//     PlcTask Outputs/GVL_iXlinker.EtherCAT_Master_EKxxxx.Beckhoff_EKx9xx.Beckhoff_EKx9xxEK1122.A_0006_EK1960_2600_0021.Module_2_FSOUT.Outputs.Relais_Module_Channel_1_Standard_Output_X4_1_X4_5 <-> Module 2 (FSOUT)/Outputs/Relais Module.Channel 1.Standard Output (X4.1, X4.5)
//     PlcTask Outputs/GVL_iXlinker.EtherCAT_Master_EKxxxx.Beckhoff_EKx9xx.Beckhoff_EKx9xxEK1122.A_0006_EK1960_2600_0021.Module_2_FSOUT.Outputs.Relais_Module_Channel_2_Standard_Output_X4_2_X4_6 <-> Module 2 (FSOUT)/Outputs/Relais Module.Channel 2.Standard Output (X4.2, X4.6)
//     PlcTask Outputs/GVL_iXlinker.EtherCAT_Master_EKxxxx.Beckhoff_EKx9xx.Beckhoff_EKx9xxEK1122.A_0006_EK1960_2600_0021.Module_2_FSOUT.Outputs.Relais_Module_Channel_3_Standard_Output_X4_3_X4_7 <-> Module 2 (FSOUT)/Outputs/Relais Module.Channel 3.Standard Output (X4.3, X4.7)
//     PlcTask Outputs/GVL_iXlinker.EtherCAT_Master_EKxxxx.Beckhoff_EKx9xx.Beckhoff_EKx9xxEK1122.A_0006_EK1960_2600_0021.Module_2_FSOUT.Outputs.Relais_Module_Channel_4_Standard_Output_X4_4_X4_8 <-> Module 2 (FSOUT)/Outputs/Relais Module.Channel 4.Standard Output (X4.4, X4.8)
//     PlcTask Inputs/GVL_iXlinker.EtherCAT_Master_EKxxxx.Beckhoff_EKx9xx.Beckhoff_EKx9xxEK1122.A_0006_EK1960_2600_0021.Module_3_FSLOGIC.FSLOGIC_Inputs.Safe_Logic_State <-> Module 3 (FSLOGIC)/FSLOGIC Inputs/Safe Logic State
//     PlcTask Inputs/GVL_iXlinker.EtherCAT_Master_EKxxxx.Beckhoff_EKx9xx.Beckhoff_EKx9xxEK1122.A_0006_EK1960_2600_0021.Module_3_FSLOGIC.FSLOGIC_Inputs.Cycle_Counter <-> Module 3 (FSLOGIC)/FSLOGIC Inputs/Cycle Counter
//     PlcTask Inputs/GVL_iXlinker.EtherCAT_Master_EKxxxx.Beckhoff_EKx9xx.Beckhoff_EKx9xxEK1122.A_0006_EK1960_2600_0021.WcState.WcState0 <-> WcState/WcState0
//     PlcTask Inputs/GVL_iXlinker.EtherCAT_Master_EKxxxx.Beckhoff_EKx9xx.Beckhoff_EKx9xxEK1122.A_0006_EK1960_2600_0021.WcState.WcState1 <-> WcState/WcState1
//     PlcTask Inputs/GVL_iXlinker.EtherCAT_Master_EKxxxx.Beckhoff_EKx9xx.Beckhoff_EKx9xxEK1122.A_0006_EK1960_2600_0021.WcState.InputToggle0 <-> WcState/InputToggle0
//     PlcTask Inputs/GVL_iXlinker.EtherCAT_Master_EKxxxx.Beckhoff_EKx9xx.Beckhoff_EKx9xxEK1122.A_0006_EK1960_2600_0021.WcState.InputToggle1 <-> WcState/InputToggle1
//     PlcTask Inputs/GVL_iXlinker.EtherCAT_Master_EKxxxx.Beckhoff_EKx9xx.Beckhoff_EKx9xxEK1122.A_0006_EK1960_2600_0021.InfoData.AdsAddr <-> InfoData/AdsAddr
//     PlcTask Inputs/GVL_iXlinker.EtherCAT_Master_EKxxxx.Beckhoff_EKx9xx.Beckhoff_EKx9xxEK1122.A_0006_EK1960_2600_0021.InfoData.State <-> InfoData/State
//   PLC/PLC Instance <-> EtherCAT Master EKxxxx/Beckhoff EKx9xx/Beckhoff EKx9xxEK1122/A_0007(EK1960-2608-0019)
//     PlcTask Inputs/GVL_iXlinker.EtherCAT_Master_EKxxxx.Beckhoff_EKx9xx.Beckhoff_EKx9xxEK1122.A_0007_EK1960_2608_0019.Module_1_FSoE.FSoE_Inputs.FSOE/FSoE_Command <-> Module 1 (FSoE)/FSoE Inputs/FSOE/FSoE Command
//     PlcTask Inputs/GVL_iXlinker.EtherCAT_Master_EKxxxx.Beckhoff_EKx9xx.Beckhoff_EKx9xxEK1122.A_0007_EK1960_2608_0019.Module_1_FSoE.FSoE_Inputs.FSOE/FSOUT_Module_1_Module_Fault <-> Module 1 (FSoE)/FSoE Inputs/FSOE/FSOUT Module 1.Module Fault
//     PlcTask Inputs/GVL_iXlinker.EtherCAT_Master_EKxxxx.Beckhoff_EKx9xx.Beckhoff_EKx9xxEK1122.A_0007_EK1960_2608_0019.Module_1_FSoE.FSoE_Inputs.FSOE/FSOUT_Module_2_Module_Fault <-> Module 1 (FSoE)/FSoE Inputs/FSOE/FSOUT Module 2.Module Fault
//     PlcTask Inputs/GVL_iXlinker.EtherCAT_Master_EKxxxx.Beckhoff_EKx9xx.Beckhoff_EKx9xxEK1122.A_0007_EK1960_2608_0019.Module_1_FSoE.FSoE_Inputs.FSOE/FSOUT_Module_3_Module_Fault <-> Module 1 (FSoE)/FSoE Inputs/FSOE/FSOUT Module 3.Module Fault
//     PlcTask Inputs/GVL_iXlinker.EtherCAT_Master_EKxxxx.Beckhoff_EKx9xx.Beckhoff_EKx9xxEK1122.A_0007_EK1960_2608_0019.Module_1_FSoE.FSoE_Inputs.FSOE/FSOUT_Module_4_Module_Fault <-> Module 1 (FSoE)/FSoE Inputs/FSOE/FSOUT Module 4.Module Fault
//     PlcTask Inputs/GVL_iXlinker.EtherCAT_Master_EKxxxx.Beckhoff_EKx9xx.Beckhoff_EKx9xxEK1122.A_0007_EK1960_2608_0019.Module_1_FSoE.FSoE_Inputs.FSOE/FSOUT_Module_5_Module_Fault <-> Module 1 (FSoE)/FSoE Inputs/FSOE/FSOUT Module 5.Module Fault
//     PlcTask Inputs/GVL_iXlinker.EtherCAT_Master_EKxxxx.Beckhoff_EKx9xx.Beckhoff_EKx9xxEK1122.A_0007_EK1960_2608_0019.Module_1_FSoE.FSoE_Inputs.FSOE/FSOUT_Module_6_Module_Fault <-> Module 1 (FSoE)/FSoE Inputs/FSOE/FSOUT Module 6.Module Fault
//     PlcTask Inputs/GVL_iXlinker.EtherCAT_Master_EKxxxx.Beckhoff_EKx9xx.Beckhoff_EKx9xxEK1122.A_0007_EK1960_2608_0019.Module_1_FSoE.FSoE_Inputs.FSOE/FSOUT_Relais_Module_Module_Fault <-> Module 1 (FSoE)/FSoE Inputs/FSOE/FSOUT Relais Module.Module Fault
//     PlcTask Inputs/GVL_iXlinker.EtherCAT_Master_EKxxxx.Beckhoff_EKx9xx.Beckhoff_EKx9xxEK1122.A_0007_EK1960_2608_0019.Module_1_FSoE.FSoE_Inputs.FSOE/FSIN_Module_1_Channel_1_Input <-> Module 1 (FSoE)/FSoE Inputs/FSOE/FSIN Module 1.Channel 1.Input
//     PlcTask Inputs/GVL_iXlinker.EtherCAT_Master_EKxxxx.Beckhoff_EKx9xx.Beckhoff_EKx9xxEK1122.A_0007_EK1960_2608_0019.Module_1_FSoE.FSoE_Inputs.FSOE/FSIN_Module_1_Channel_2_Input <-> Module 1 (FSoE)/FSoE Inputs/FSOE/FSIN Module 1.Channel 2.Input
//     PlcTask Inputs/GVL_iXlinker.EtherCAT_Master_EKxxxx.Beckhoff_EKx9xx.Beckhoff_EKx9xxEK1122.A_0007_EK1960_2608_0019.Module_1_FSoE.FSoE_Inputs.FSOE/FSIN_Module_2_Channel_1_Input <-> Module 1 (FSoE)/FSoE Inputs/FSOE/FSIN Module 2.Channel 1.Input
//     PlcTask Inputs/GVL_iXlinker.EtherCAT_Master_EKxxxx.Beckhoff_EKx9xx.Beckhoff_EKx9xxEK1122.A_0007_EK1960_2608_0019.Module_1_FSoE.FSoE_Inputs.FSOE/FSIN_Module_2_Channel_2_Input <-> Module 1 (FSoE)/FSoE Inputs/FSOE/FSIN Module 2.Channel 2.Input
//     PlcTask Inputs/GVL_iXlinker.EtherCAT_Master_EKxxxx.Beckhoff_EKx9xx.Beckhoff_EKx9xxEK1122.A_0007_EK1960_2608_0019.Module_1_FSoE.FSoE_Inputs.FSOE/FSIN_Module_3_Channel_1_Input <-> Module 1 (FSoE)/FSoE Inputs/FSOE/FSIN Module 3.Channel 1.Input
//     PlcTask Inputs/GVL_iXlinker.EtherCAT_Master_EKxxxx.Beckhoff_EKx9xx.Beckhoff_EKx9xxEK1122.A_0007_EK1960_2608_0019.Module_1_FSoE.FSoE_Inputs.FSOE/FSIN_Module_3_Channel_2_Input <-> Module 1 (FSoE)/FSoE Inputs/FSOE/FSIN Module 3.Channel 2.Input
//     PlcTask Inputs/GVL_iXlinker.EtherCAT_Master_EKxxxx.Beckhoff_EKx9xx.Beckhoff_EKx9xxEK1122.A_0007_EK1960_2608_0019.Module_1_FSoE.FSoE_Inputs.FSOE/FSIN_Module_4_Channel_1_Input <-> Module 1 (FSoE)/FSoE Inputs/FSOE/FSIN Module 4.Channel 1.Input
//     PlcTask Inputs/GVL_iXlinker.EtherCAT_Master_EKxxxx.Beckhoff_EKx9xx.Beckhoff_EKx9xxEK1122.A_0007_EK1960_2608_0019.Module_1_FSoE.FSoE_Inputs.FSOE/FSIN_Module_4_Channel_2_Input <-> Module 1 (FSoE)/FSoE Inputs/FSOE/FSIN Module 4.Channel 2.Input
//     PlcTask Inputs/GVL_iXlinker.EtherCAT_Master_EKxxxx.Beckhoff_EKx9xx.Beckhoff_EKx9xxEK1122.A_0007_EK1960_2608_0019.Module_1_FSoE.FSoE_Inputs.FSOE/FSIN_Module_5_Channel_1_Input <-> Module 1 (FSoE)/FSoE Inputs/FSOE/FSIN Module 5.Channel 1.Input
//     PlcTask Inputs/GVL_iXlinker.EtherCAT_Master_EKxxxx.Beckhoff_EKx9xx.Beckhoff_EKx9xxEK1122.A_0007_EK1960_2608_0019.Module_1_FSoE.FSoE_Inputs.FSOE/FSIN_Module_5_Channel_2_Input <-> Module 1 (FSoE)/FSoE Inputs/FSOE/FSIN Module 5.Channel 2.Input
//     PlcTask Inputs/GVL_iXlinker.EtherCAT_Master_EKxxxx.Beckhoff_EKx9xx.Beckhoff_EKx9xxEK1122.A_0007_EK1960_2608_0019.Module_1_FSoE.FSoE_Inputs.FSOE/FSIN_Module_6_Channel_1_Input <-> Module 1 (FSoE)/FSoE Inputs/FSOE/FSIN Module 6.Channel 1.Input
//     PlcTask Inputs/GVL_iXlinker.EtherCAT_Master_EKxxxx.Beckhoff_EKx9xx.Beckhoff_EKx9xxEK1122.A_0007_EK1960_2608_0019.Module_1_FSoE.FSoE_Inputs.FSOE/FSIN_Module_6_Channel_2_Input <-> Module 1 (FSoE)/FSoE Inputs/FSOE/FSIN Module 6.Channel 2.Input
//     PlcTask Inputs/GVL_iXlinker.EtherCAT_Master_EKxxxx.Beckhoff_EKx9xx.Beckhoff_EKx9xxEK1122.A_0007_EK1960_2608_0019.Module_1_FSoE.FSoE_Inputs.FSOE/FSIN_Module_7_Channel_1_Input <-> Module 1 (FSoE)/FSoE Inputs/FSOE/FSIN Module 7.Channel 1.Input
//     PlcTask Inputs/GVL_iXlinker.EtherCAT_Master_EKxxxx.Beckhoff_EKx9xx.Beckhoff_EKx9xxEK1122.A_0007_EK1960_2608_0019.Module_1_FSoE.FSoE_Inputs.FSOE/FSIN_Module_7_Channel_2_Input <-> Module 1 (FSoE)/FSoE Inputs/FSOE/FSIN Module 7.Channel 2.Input
//     PlcTask Inputs/GVL_iXlinker.EtherCAT_Master_EKxxxx.Beckhoff_EKx9xx.Beckhoff_EKx9xxEK1122.A_0007_EK1960_2608_0019.Module_1_FSoE.FSoE_Inputs.FSOE/FSIN_Module_8_Channel_1_Input <-> Module 1 (FSoE)/FSoE Inputs/FSOE/FSIN Module 8.Channel 1.Input
//     PlcTask Inputs/GVL_iXlinker.EtherCAT_Master_EKxxxx.Beckhoff_EKx9xx.Beckhoff_EKx9xxEK1122.A_0007_EK1960_2608_0019.Module_1_FSoE.FSoE_Inputs.FSOE/FSIN_Module_8_Channel_2_Input <-> Module 1 (FSoE)/FSoE Inputs/FSOE/FSIN Module 8.Channel 2.Input
//     PlcTask Inputs/GVL_iXlinker.EtherCAT_Master_EKxxxx.Beckhoff_EKx9xx.Beckhoff_EKx9xxEK1122.A_0007_EK1960_2608_0019.Module_1_FSoE.FSoE_Inputs.FSOE/FSIN_Module_9_Channel_1_Input <-> Module 1 (FSoE)/FSoE Inputs/FSOE/FSIN Module 9.Channel 1.Input
//     PlcTask Inputs/GVL_iXlinker.EtherCAT_Master_EKxxxx.Beckhoff_EKx9xx.Beckhoff_EKx9xxEK1122.A_0007_EK1960_2608_0019.Module_1_FSoE.FSoE_Inputs.FSOE/FSIN_Module_9_Channel_2_Input <-> Module 1 (FSoE)/FSoE Inputs/FSOE/FSIN Module 9.Channel 2.Input
//     PlcTask Inputs/GVL_iXlinker.EtherCAT_Master_EKxxxx.Beckhoff_EKx9xx.Beckhoff_EKx9xxEK1122.A_0007_EK1960_2608_0019.Module_1_FSoE.FSoE_Inputs.FSOE/FSIN_Module_10_Channel_1_Input <-> Module 1 (FSoE)/FSoE Inputs/FSOE/FSIN Module 10.Channel 1.Input
//     PlcTask Inputs/GVL_iXlinker.EtherCAT_Master_EKxxxx.Beckhoff_EKx9xx.Beckhoff_EKx9xxEK1122.A_0007_EK1960_2608_0019.Module_1_FSoE.FSoE_Inputs.FSOE/FSIN_Module_10_Channel_2_Input <-> Module 1 (FSoE)/FSoE Inputs/FSOE/FSIN Module 10.Channel 2.Input
//     PlcTask Inputs/GVL_iXlinker.EtherCAT_Master_EKxxxx.Beckhoff_EKx9xx.Beckhoff_EKx9xxEK1122.A_0007_EK1960_2608_0019.Module_1_FSoE.FSoE_Inputs.FSOE/FSIN_Module_1_Module_Fault <-> Module 1 (FSoE)/FSoE Inputs/FSOE/FSIN Module 1.Module Fault
//     PlcTask Inputs/GVL_iXlinker.EtherCAT_Master_EKxxxx.Beckhoff_EKx9xx.Beckhoff_EKx9xxEK1122.A_0007_EK1960_2608_0019.Module_1_FSoE.FSoE_Inputs.FSOE/FSIN_Module_2_Module_Fault <-> Module 1 (FSoE)/FSoE Inputs/FSOE/FSIN Module 2.Module Fault
//     PlcTask Inputs/GVL_iXlinker.EtherCAT_Master_EKxxxx.Beckhoff_EKx9xx.Beckhoff_EKx9xxEK1122.A_0007_EK1960_2608_0019.Module_1_FSoE.FSoE_Inputs.FSOE/FSIN_Module_3_Module_Fault <-> Module 1 (FSoE)/FSoE Inputs/FSOE/FSIN Module 3.Module Fault
//     PlcTask Inputs/GVL_iXlinker.EtherCAT_Master_EKxxxx.Beckhoff_EKx9xx.Beckhoff_EKx9xxEK1122.A_0007_EK1960_2608_0019.Module_1_FSoE.FSoE_Inputs.FSOE/FSIN_Module_4_Module_Fault <-> Module 1 (FSoE)/FSoE Inputs/FSOE/FSIN Module 4.Module Fault
//     PlcTask Inputs/GVL_iXlinker.EtherCAT_Master_EKxxxx.Beckhoff_EKx9xx.Beckhoff_EKx9xxEK1122.A_0007_EK1960_2608_0019.Module_1_FSoE.FSoE_Inputs.FSOE/FSIN_Module_5_Module_Fault <-> Module 1 (FSoE)/FSoE Inputs/FSOE/FSIN Module 5.Module Fault
//     PlcTask Inputs/GVL_iXlinker.EtherCAT_Master_EKxxxx.Beckhoff_EKx9xx.Beckhoff_EKx9xxEK1122.A_0007_EK1960_2608_0019.Module_1_FSoE.FSoE_Inputs.FSOE/FSIN_Module_6_Module_Fault <-> Module 1 (FSoE)/FSoE Inputs/FSOE/FSIN Module 6.Module Fault
//     PlcTask Inputs/GVL_iXlinker.EtherCAT_Master_EKxxxx.Beckhoff_EKx9xx.Beckhoff_EKx9xxEK1122.A_0007_EK1960_2608_0019.Module_1_FSoE.FSoE_Inputs.FSOE/FSIN_Module_7_Module_Fault <-> Module 1 (FSoE)/FSoE Inputs/FSOE/FSIN Module 7.Module Fault
//     PlcTask Inputs/GVL_iXlinker.EtherCAT_Master_EKxxxx.Beckhoff_EKx9xx.Beckhoff_EKx9xxEK1122.A_0007_EK1960_2608_0019.Module_1_FSoE.FSoE_Inputs.FSOE/FSIN_Module_8_Module_Fault <-> Module 1 (FSoE)/FSoE Inputs/FSOE/FSIN Module 8.Module Fault
//     PlcTask Inputs/GVL_iXlinker.EtherCAT_Master_EKxxxx.Beckhoff_EKx9xx.Beckhoff_EKx9xxEK1122.A_0007_EK1960_2608_0019.Module_1_FSoE.FSoE_Inputs.FSOE/FSoE_CRC_000 <-> Module 1 (FSoE)/FSoE Inputs/FSOE/FSoE CRC 000
//     PlcTask Inputs/GVL_iXlinker.EtherCAT_Master_EKxxxx.Beckhoff_EKx9xx.Beckhoff_EKx9xxEK1122.A_0007_EK1960_2608_0019.Module_1_FSoE.FSoE_Inputs.FSOE/FSoE_CRC_001 <-> Module 1 (FSoE)/FSoE Inputs/FSOE/FSoE CRC 001
//     PlcTask Inputs/GVL_iXlinker.EtherCAT_Master_EKxxxx.Beckhoff_EKx9xx.Beckhoff_EKx9xxEK1122.A_0007_EK1960_2608_0019.Module_1_FSoE.FSoE_Inputs.FSOE/FSoE_CRC_002 <-> Module 1 (FSoE)/FSoE Inputs/FSOE/FSoE CRC 002
//     PlcTask Inputs/GVL_iXlinker.EtherCAT_Master_EKxxxx.Beckhoff_EKx9xx.Beckhoff_EKx9xxEK1122.A_0007_EK1960_2608_0019.Module_1_FSoE.FSoE_Inputs.FSOE/FSIN_Module_9_Module_Fault_1 <-> Module 1 (FSoE)/FSoE Inputs/FSOE/FSIN Module 9.Module Fault 1
//     PlcTask Inputs/GVL_iXlinker.EtherCAT_Master_EKxxxx.Beckhoff_EKx9xx.Beckhoff_EKx9xxEK1122.A_0007_EK1960_2608_0019.Module_1_FSoE.FSoE_Inputs.FSOE/FSIN_Module_9_Module_Fault_2 <-> Module 1 (FSoE)/FSoE Inputs/FSOE/FSIN Module 9.Module Fault 2
//     PlcTask Inputs/GVL_iXlinker.EtherCAT_Master_EKxxxx.Beckhoff_EKx9xx.Beckhoff_EKx9xxEK1122.A_0007_EK1960_2608_0019.Module_1_FSoE.FSoE_Inputs.FSOE/FSIN_Module_10_Module_Fault_1 <-> Module 1 (FSoE)/FSoE Inputs/FSOE/FSIN Module 10.Module Fault 1
//     PlcTask Inputs/GVL_iXlinker.EtherCAT_Master_EKxxxx.Beckhoff_EKx9xx.Beckhoff_EKx9xxEK1122.A_0007_EK1960_2608_0019.Module_1_FSoE.FSoE_Inputs.FSOE/FSIN_Module_10_Module_Fault_2 <-> Module 1 (FSoE)/FSoE Inputs/FSOE/FSIN Module 10.Module Fault 2
//     PlcTask Inputs/GVL_iXlinker.EtherCAT_Master_EKxxxx.Beckhoff_EKx9xx.Beckhoff_EKx9xxEK1122.A_0007_EK1960_2608_0019.Module_1_FSoE.FSoE_Inputs.FSOE/FSoE_Connection_ID <-> Module 1 (FSoE)/FSoE Inputs/FSOE/FSoE Connection ID
//     PlcTask Outputs/GVL_iXlinker.EtherCAT_Master_EKxxxx.Beckhoff_EKx9xx.Beckhoff_EKx9xxEK1122.A_0007_EK1960_2608_0019.Module_1_FSoE.FSoE_Outputs.FSOE/FSoE_Command <-> Module 1 (FSoE)/FSoE Outputs/FSOE/FSoE Command
//     PlcTask Outputs/GVL_iXlinker.EtherCAT_Master_EKxxxx.Beckhoff_EKx9xx.Beckhoff_EKx9xxEK1122.A_0007_EK1960_2608_0019.Module_1_FSoE.FSoE_Outputs.FSOE/FSOUT_Module_1_Channel_1_Output <-> Module 1 (FSoE)/FSoE Outputs/FSOE/FSOUT Module 1.Channel 1.Output
//     PlcTask Outputs/GVL_iXlinker.EtherCAT_Master_EKxxxx.Beckhoff_EKx9xx.Beckhoff_EKx9xxEK1122.A_0007_EK1960_2608_0019.Module_1_FSoE.FSoE_Outputs.FSOE/FSOUT_Module_1_Channel_2_Output <-> Module 1 (FSoE)/FSoE Outputs/FSOE/FSOUT Module 1.Channel 2.Output
//     PlcTask Outputs/GVL_iXlinker.EtherCAT_Master_EKxxxx.Beckhoff_EKx9xx.Beckhoff_EKx9xxEK1122.A_0007_EK1960_2608_0019.Module_1_FSoE.FSoE_Outputs.FSOE/FSOUT_Module_1_Channel_3_Output <-> Module 1 (FSoE)/FSoE Outputs/FSOE/FSOUT Module 1.Channel 3.Output
//     PlcTask Outputs/GVL_iXlinker.EtherCAT_Master_EKxxxx.Beckhoff_EKx9xx.Beckhoff_EKx9xxEK1122.A_0007_EK1960_2608_0019.Module_1_FSoE.FSoE_Outputs.FSOE/FSOUT_Module_1_Channel_4_Output <-> Module 1 (FSoE)/FSoE Outputs/FSOE/FSOUT Module 1.Channel 4.Output
//     PlcTask Outputs/GVL_iXlinker.EtherCAT_Master_EKxxxx.Beckhoff_EKx9xx.Beckhoff_EKx9xxEK1122.A_0007_EK1960_2608_0019.Module_1_FSoE.FSoE_Outputs.FSOE/FSOUT_Module_2_Channel_1_Output <-> Module 1 (FSoE)/FSoE Outputs/FSOE/FSOUT Module 2.Channel 1.Output
//     PlcTask Outputs/GVL_iXlinker.EtherCAT_Master_EKxxxx.Beckhoff_EKx9xx.Beckhoff_EKx9xxEK1122.A_0007_EK1960_2608_0019.Module_1_FSoE.FSoE_Outputs.FSOE/FSOUT_Module_2_Channel_2_Output <-> Module 1 (FSoE)/FSoE Outputs/FSOE/FSOUT Module 2.Channel 2.Output
//     PlcTask Outputs/GVL_iXlinker.EtherCAT_Master_EKxxxx.Beckhoff_EKx9xx.Beckhoff_EKx9xxEK1122.A_0007_EK1960_2608_0019.Module_1_FSoE.FSoE_Outputs.FSOE/FSOUT_Module_2_Channel_3_Output <-> Module 1 (FSoE)/FSoE Outputs/FSOE/FSOUT Module 2.Channel 3.Output
//     PlcTask Outputs/GVL_iXlinker.EtherCAT_Master_EKxxxx.Beckhoff_EKx9xx.Beckhoff_EKx9xxEK1122.A_0007_EK1960_2608_0019.Module_1_FSoE.FSoE_Outputs.FSOE/FSOUT_Module_2_Channel_4_Output <-> Module 1 (FSoE)/FSoE Outputs/FSOE/FSOUT Module 2.Channel 4.Output
//     PlcTask Outputs/GVL_iXlinker.EtherCAT_Master_EKxxxx.Beckhoff_EKx9xx.Beckhoff_EKx9xxEK1122.A_0007_EK1960_2608_0019.Module_1_FSoE.FSoE_Outputs.FSOE/FSOUT_Module_3_Channel_1_Output <-> Module 1 (FSoE)/FSoE Outputs/FSOE/FSOUT Module 3.Channel 1.Output
//     PlcTask Outputs/GVL_iXlinker.EtherCAT_Master_EKxxxx.Beckhoff_EKx9xx.Beckhoff_EKx9xxEK1122.A_0007_EK1960_2608_0019.Module_1_FSoE.FSoE_Outputs.FSOE/FSOUT_Module_3_Channel_2_Output <-> Module 1 (FSoE)/FSoE Outputs/FSOE/FSOUT Module 3.Channel 2.Output
//     PlcTask Outputs/GVL_iXlinker.EtherCAT_Master_EKxxxx.Beckhoff_EKx9xx.Beckhoff_EKx9xxEK1122.A_0007_EK1960_2608_0019.Module_1_FSoE.FSoE_Outputs.FSOE/FSOUT_Module_3_Channel_3_Output <-> Module 1 (FSoE)/FSoE Outputs/FSOE/FSOUT Module 3.Channel 3.Output
//     PlcTask Outputs/GVL_iXlinker.EtherCAT_Master_EKxxxx.Beckhoff_EKx9xx.Beckhoff_EKx9xxEK1122.A_0007_EK1960_2608_0019.Module_1_FSoE.FSoE_Outputs.FSOE/FSOUT_Module_3_Channel_4_Output <-> Module 1 (FSoE)/FSoE Outputs/FSOE/FSOUT Module 3.Channel 4.Output
//     PlcTask Outputs/GVL_iXlinker.EtherCAT_Master_EKxxxx.Beckhoff_EKx9xx.Beckhoff_EKx9xxEK1122.A_0007_EK1960_2608_0019.Module_1_FSoE.FSoE_Outputs.FSOE/FSOUT_Module_4_Channel_1_Output <-> Module 1 (FSoE)/FSoE Outputs/FSOE/FSOUT Module 4.Channel 1.Output
//     PlcTask Outputs/GVL_iXlinker.EtherCAT_Master_EKxxxx.Beckhoff_EKx9xx.Beckhoff_EKx9xxEK1122.A_0007_EK1960_2608_0019.Module_1_FSoE.FSoE_Outputs.FSOE/FSOUT_Module_4_Channel_2_Output <-> Module 1 (FSoE)/FSoE Outputs/FSOE/FSOUT Module 4.Channel 2.Output
//     PlcTask Outputs/GVL_iXlinker.EtherCAT_Master_EKxxxx.Beckhoff_EKx9xx.Beckhoff_EKx9xxEK1122.A_0007_EK1960_2608_0019.Module_1_FSoE.FSoE_Outputs.FSOE/FSOUT_Module_4_Channel_3_Output <-> Module 1 (FSoE)/FSoE Outputs/FSOE/FSOUT Module 4.Channel 3.Output
//     PlcTask Outputs/GVL_iXlinker.EtherCAT_Master_EKxxxx.Beckhoff_EKx9xx.Beckhoff_EKx9xxEK1122.A_0007_EK1960_2608_0019.Module_1_FSoE.FSoE_Outputs.FSOE/FSOUT_Module_4_Channel_4_Output <-> Module 1 (FSoE)/FSoE Outputs/FSOE/FSOUT Module 4.Channel 4.Output
//     PlcTask Outputs/GVL_iXlinker.EtherCAT_Master_EKxxxx.Beckhoff_EKx9xx.Beckhoff_EKx9xxEK1122.A_0007_EK1960_2608_0019.Module_1_FSoE.FSoE_Outputs.FSOE/FSOUT_Module_5_Channel_1_Output <-> Module 1 (FSoE)/FSoE Outputs/FSOE/FSOUT Module 5.Channel 1.Output
//     PlcTask Outputs/GVL_iXlinker.EtherCAT_Master_EKxxxx.Beckhoff_EKx9xx.Beckhoff_EKx9xxEK1122.A_0007_EK1960_2608_0019.Module_1_FSoE.FSoE_Outputs.FSOE/FSOUT_Module_5_Channel_2_Output <-> Module 1 (FSoE)/FSoE Outputs/FSOE/FSOUT Module 5.Channel 2.Output
//     PlcTask Outputs/GVL_iXlinker.EtherCAT_Master_EKxxxx.Beckhoff_EKx9xx.Beckhoff_EKx9xxEK1122.A_0007_EK1960_2608_0019.Module_1_FSoE.FSoE_Outputs.FSOE/FSOUT_Module_5_Channel_3_Output <-> Module 1 (FSoE)/FSoE Outputs/FSOE/FSOUT Module 5.Channel 3.Output
//     PlcTask Outputs/GVL_iXlinker.EtherCAT_Master_EKxxxx.Beckhoff_EKx9xx.Beckhoff_EKx9xxEK1122.A_0007_EK1960_2608_0019.Module_1_FSoE.FSoE_Outputs.FSOE/FSOUT_Module_5_Channel_4_Output <-> Module 1 (FSoE)/FSoE Outputs/FSOE/FSOUT Module 5.Channel 4.Output
//     PlcTask Outputs/GVL_iXlinker.EtherCAT_Master_EKxxxx.Beckhoff_EKx9xx.Beckhoff_EKx9xxEK1122.A_0007_EK1960_2608_0019.Module_1_FSoE.FSoE_Outputs.FSOE/FSOUT_Module_6_Channel_1_Output <-> Module 1 (FSoE)/FSoE Outputs/FSOE/FSOUT Module 6.Channel 1.Output
//     PlcTask Outputs/GVL_iXlinker.EtherCAT_Master_EKxxxx.Beckhoff_EKx9xx.Beckhoff_EKx9xxEK1122.A_0007_EK1960_2608_0019.Module_1_FSoE.FSoE_Outputs.FSOE/FSOUT_Module_6_Channel_2_Output <-> Module 1 (FSoE)/FSoE Outputs/FSOE/FSOUT Module 6.Channel 2.Output
//     PlcTask Outputs/GVL_iXlinker.EtherCAT_Master_EKxxxx.Beckhoff_EKx9xx.Beckhoff_EKx9xxEK1122.A_0007_EK1960_2608_0019.Module_1_FSoE.FSoE_Outputs.FSOE/FSOUT_Module_6_Channel_3_Output <-> Module 1 (FSoE)/FSoE Outputs/FSOE/FSOUT Module 6.Channel 3.Output
//     PlcTask Outputs/GVL_iXlinker.EtherCAT_Master_EKxxxx.Beckhoff_EKx9xx.Beckhoff_EKx9xxEK1122.A_0007_EK1960_2608_0019.Module_1_FSoE.FSoE_Outputs.FSOE/FSOUT_Module_6_Channel_4_Output <-> Module 1 (FSoE)/FSoE Outputs/FSOE/FSOUT Module 6.Channel 4.Output
//     PlcTask Outputs/GVL_iXlinker.EtherCAT_Master_EKxxxx.Beckhoff_EKx9xx.Beckhoff_EKx9xxEK1122.A_0007_EK1960_2608_0019.Module_1_FSoE.FSoE_Outputs.FSOE/FSOUT_Module_1_ErrAck <-> Module 1 (FSoE)/FSoE Outputs/FSOE/FSOUT Module 1.ErrAck
//     PlcTask Outputs/GVL_iXlinker.EtherCAT_Master_EKxxxx.Beckhoff_EKx9xx.Beckhoff_EKx9xxEK1122.A_0007_EK1960_2608_0019.Module_1_FSoE.FSoE_Outputs.FSOE/FSOUT_Module_2_ErrAck <-> Module 1 (FSoE)/FSoE Outputs/FSOE/FSOUT Module 2.ErrAck
//     PlcTask Outputs/GVL_iXlinker.EtherCAT_Master_EKxxxx.Beckhoff_EKx9xx.Beckhoff_EKx9xxEK1122.A_0007_EK1960_2608_0019.Module_1_FSoE.FSoE_Outputs.FSOE/FSOUT_Module_3_ErrAck <-> Module 1 (FSoE)/FSoE Outputs/FSOE/FSOUT Module 3.ErrAck
//     PlcTask Outputs/GVL_iXlinker.EtherCAT_Master_EKxxxx.Beckhoff_EKx9xx.Beckhoff_EKx9xxEK1122.A_0007_EK1960_2608_0019.Module_1_FSoE.FSoE_Outputs.FSOE/FSOUT_Module_4_ErrAck <-> Module 1 (FSoE)/FSoE Outputs/FSOE/FSOUT Module 4.ErrAck
//     PlcTask Outputs/GVL_iXlinker.EtherCAT_Master_EKxxxx.Beckhoff_EKx9xx.Beckhoff_EKx9xxEK1122.A_0007_EK1960_2608_0019.Module_1_FSoE.FSoE_Outputs.FSOE/FSOUT_Module_5_ErrAck <-> Module 1 (FSoE)/FSoE Outputs/FSOE/FSOUT Module 5.ErrAck
//     PlcTask Outputs/GVL_iXlinker.EtherCAT_Master_EKxxxx.Beckhoff_EKx9xx.Beckhoff_EKx9xxEK1122.A_0007_EK1960_2608_0019.Module_1_FSoE.FSoE_Outputs.FSOE/FSOUT_Module_6_ErrAck <-> Module 1 (FSoE)/FSoE Outputs/FSOE/FSOUT Module 6.ErrAck
//     PlcTask Outputs/GVL_iXlinker.EtherCAT_Master_EKxxxx.Beckhoff_EKx9xx.Beckhoff_EKx9xxEK1122.A_0007_EK1960_2608_0019.Module_1_FSoE.FSoE_Outputs.FSOE/FSoE_CRC_000 <-> Module 1 (FSoE)/FSoE Outputs/FSOE/FSoE CRC 000
//     PlcTask Outputs/GVL_iXlinker.EtherCAT_Master_EKxxxx.Beckhoff_EKx9xx.Beckhoff_EKx9xxEK1122.A_0007_EK1960_2608_0019.Module_1_FSoE.FSoE_Outputs.FSOE/FSoE_CRC_001 <-> Module 1 (FSoE)/FSoE Outputs/FSOE/FSoE CRC 001
//     PlcTask Outputs/GVL_iXlinker.EtherCAT_Master_EKxxxx.Beckhoff_EKx9xx.Beckhoff_EKx9xxEK1122.A_0007_EK1960_2608_0019.Module_1_FSoE.FSoE_Outputs.FSOE/FSoE_CRC_002 <-> Module 1 (FSoE)/FSoE Outputs/FSOE/FSoE CRC 002
//     PlcTask Outputs/GVL_iXlinker.EtherCAT_Master_EKxxxx.Beckhoff_EKx9xx.Beckhoff_EKx9xxEK1122.A_0007_EK1960_2608_0019.Module_1_FSoE.FSoE_Outputs.FSOE/FSOUT_Relais_Module_Channel_1_Output <-> Module 1 (FSoE)/FSoE Outputs/FSOE/FSOUT Relais Module.Channel 1.Output
//     PlcTask Outputs/GVL_iXlinker.EtherCAT_Master_EKxxxx.Beckhoff_EKx9xx.Beckhoff_EKx9xxEK1122.A_0007_EK1960_2608_0019.Module_1_FSoE.FSoE_Outputs.FSOE/FSOUT_Relais_Module_Channel_2_Output <-> Module 1 (FSoE)/FSoE Outputs/FSOE/FSOUT Relais Module.Channel 2.Output
//     PlcTask Outputs/GVL_iXlinker.EtherCAT_Master_EKxxxx.Beckhoff_EKx9xx.Beckhoff_EKx9xxEK1122.A_0007_EK1960_2608_0019.Module_1_FSoE.FSoE_Outputs.FSOE/FSOUT_Relais_Module_Channel_3_Output <-> Module 1 (FSoE)/FSoE Outputs/FSOE/FSOUT Relais Module.Channel 3.Output
//     PlcTask Outputs/GVL_iXlinker.EtherCAT_Master_EKxxxx.Beckhoff_EKx9xx.Beckhoff_EKx9xxEK1122.A_0007_EK1960_2608_0019.Module_1_FSoE.FSoE_Outputs.FSOE/FSOUT_Relais_Module_Channel_4_Output <-> Module 1 (FSoE)/FSoE Outputs/FSOE/FSOUT Relais Module.Channel 4.Output
//     PlcTask Outputs/GVL_iXlinker.EtherCAT_Master_EKxxxx.Beckhoff_EKx9xx.Beckhoff_EKx9xxEK1122.A_0007_EK1960_2608_0019.Module_1_FSoE.FSoE_Outputs.FSOE/FSOUT_Relais_Module_ErrAck <-> Module 1 (FSoE)/FSoE Outputs/FSOE/FSOUT Relais Module.ErrAck
//     PlcTask Outputs/GVL_iXlinker.EtherCAT_Master_EKxxxx.Beckhoff_EKx9xx.Beckhoff_EKx9xxEK1122.A_0007_EK1960_2608_0019.Module_1_FSoE.FSoE_Outputs.FSOE/FSIN_Module_1_ErrAck <-> Module 1 (FSoE)/FSoE Outputs/FSOE/FSIN Module 1.ErrAck
//     PlcTask Outputs/GVL_iXlinker.EtherCAT_Master_EKxxxx.Beckhoff_EKx9xx.Beckhoff_EKx9xxEK1122.A_0007_EK1960_2608_0019.Module_1_FSoE.FSoE_Outputs.FSOE/FSIN_Module_2_ErrAck <-> Module 1 (FSoE)/FSoE Outputs/FSOE/FSIN Module 2.ErrAck
//     PlcTask Outputs/GVL_iXlinker.EtherCAT_Master_EKxxxx.Beckhoff_EKx9xx.Beckhoff_EKx9xxEK1122.A_0007_EK1960_2608_0019.Module_1_FSoE.FSoE_Outputs.FSOE/FSIN_Module_3_ErrAck <-> Module 1 (FSoE)/FSoE Outputs/FSOE/FSIN Module 3.ErrAck
//     PlcTask Outputs/GVL_iXlinker.EtherCAT_Master_EKxxxx.Beckhoff_EKx9xx.Beckhoff_EKx9xxEK1122.A_0007_EK1960_2608_0019.Module_1_FSoE.FSoE_Outputs.FSOE/FSIN_Module_4_ErrAck <-> Module 1 (FSoE)/FSoE Outputs/FSOE/FSIN Module 4.ErrAck
//     PlcTask Outputs/GVL_iXlinker.EtherCAT_Master_EKxxxx.Beckhoff_EKx9xx.Beckhoff_EKx9xxEK1122.A_0007_EK1960_2608_0019.Module_1_FSoE.FSoE_Outputs.FSOE/FSIN_Module_5_ErrAck <-> Module 1 (FSoE)/FSoE Outputs/FSOE/FSIN Module 5.ErrAck
//     PlcTask Outputs/GVL_iXlinker.EtherCAT_Master_EKxxxx.Beckhoff_EKx9xx.Beckhoff_EKx9xxEK1122.A_0007_EK1960_2608_0019.Module_1_FSoE.FSoE_Outputs.FSOE/FSIN_Module_6_ErrAck <-> Module 1 (FSoE)/FSoE Outputs/FSOE/FSIN Module 6.ErrAck
//     PlcTask Outputs/GVL_iXlinker.EtherCAT_Master_EKxxxx.Beckhoff_EKx9xx.Beckhoff_EKx9xxEK1122.A_0007_EK1960_2608_0019.Module_1_FSoE.FSoE_Outputs.FSOE/FSIN_Module_7_ErrAck <-> Module 1 (FSoE)/FSoE Outputs/FSOE/FSIN Module 7.ErrAck
//     PlcTask Outputs/GVL_iXlinker.EtherCAT_Master_EKxxxx.Beckhoff_EKx9xx.Beckhoff_EKx9xxEK1122.A_0007_EK1960_2608_0019.Module_1_FSoE.FSoE_Outputs.FSOE/FSIN_Module_8_ErrAck <-> Module 1 (FSoE)/FSoE Outputs/FSOE/FSIN Module 8.ErrAck
//     PlcTask Outputs/GVL_iXlinker.EtherCAT_Master_EKxxxx.Beckhoff_EKx9xx.Beckhoff_EKx9xxEK1122.A_0007_EK1960_2608_0019.Module_1_FSoE.FSoE_Outputs.FSOE/FSIN_Module_9_ErrAck_1 <-> Module 1 (FSoE)/FSoE Outputs/FSOE/FSIN Module 9.ErrAck 1
//     PlcTask Outputs/GVL_iXlinker.EtherCAT_Master_EKxxxx.Beckhoff_EKx9xx.Beckhoff_EKx9xxEK1122.A_0007_EK1960_2608_0019.Module_1_FSoE.FSoE_Outputs.FSOE/FSIN_Module_9_ErrAck_2 <-> Module 1 (FSoE)/FSoE Outputs/FSOE/FSIN Module 9.ErrAck 2
//     PlcTask Outputs/GVL_iXlinker.EtherCAT_Master_EKxxxx.Beckhoff_EKx9xx.Beckhoff_EKx9xxEK1122.A_0007_EK1960_2608_0019.Module_1_FSoE.FSoE_Outputs.FSOE/FSIN_Module_10_ErrAck_1 <-> Module 1 (FSoE)/FSoE Outputs/FSOE/FSIN Module 10.ErrAck 1
//     PlcTask Outputs/GVL_iXlinker.EtherCAT_Master_EKxxxx.Beckhoff_EKx9xx.Beckhoff_EKx9xxEK1122.A_0007_EK1960_2608_0019.Module_1_FSoE.FSoE_Outputs.FSOE/FSIN_Module_10_ErrAck_2 <-> Module 1 (FSoE)/FSoE Outputs/FSOE/FSIN Module 10.ErrAck 2
//     PlcTask Outputs/GVL_iXlinker.EtherCAT_Master_EKxxxx.Beckhoff_EKx9xx.Beckhoff_EKx9xxEK1122.A_0007_EK1960_2608_0019.Module_1_FSoE.FSoE_Outputs.FSOE/FSoE_Connection_ID <-> Module 1 (FSoE)/FSoE Outputs/FSOE/FSoE Connection ID
//     PlcTask Outputs/GVL_iXlinker.EtherCAT_Master_EKxxxx.Beckhoff_EKx9xx.Beckhoff_EKx9xxEK1122.A_0007_EK1960_2608_0019.Module_2_FSOUT.Outputs.Module_1_Channel_1_Standard_Output_X5_1 <-> Module 2 (FSOUT)/Outputs/Module 1.Channel 1.Standard Output (X5.1)
//     PlcTask Outputs/GVL_iXlinker.EtherCAT_Master_EKxxxx.Beckhoff_EKx9xx.Beckhoff_EKx9xxEK1122.A_0007_EK1960_2608_0019.Module_2_FSOUT.Outputs.Module_1_Channel_2_Standard_Output_X5_2 <-> Module 2 (FSOUT)/Outputs/Module 1.Channel 2.Standard Output (X5.2)
//     PlcTask Outputs/GVL_iXlinker.EtherCAT_Master_EKxxxx.Beckhoff_EKx9xx.Beckhoff_EKx9xxEK1122.A_0007_EK1960_2608_0019.Module_2_FSOUT.Outputs.Module_1_Channel_3_Standard_Output_X5_3 <-> Module 2 (FSOUT)/Outputs/Module 1.Channel 3.Standard Output (X5.3)
//     PlcTask Outputs/GVL_iXlinker.EtherCAT_Master_EKxxxx.Beckhoff_EKx9xx.Beckhoff_EKx9xxEK1122.A_0007_EK1960_2608_0019.Module_2_FSOUT.Outputs.Module_1_Channel_4_Standard_Output_X5_4 <-> Module 2 (FSOUT)/Outputs/Module 1.Channel 4.Standard Output (X5.4)
//     PlcTask Outputs/GVL_iXlinker.EtherCAT_Master_EKxxxx.Beckhoff_EKx9xx.Beckhoff_EKx9xxEK1122.A_0007_EK1960_2608_0019.Module_2_FSOUT.Outputs.Module_2_Channel_1_Standard_Output_X5_5 <-> Module 2 (FSOUT)/Outputs/Module 2.Channel 1.Standard Output (X5.5)
//     PlcTask Outputs/GVL_iXlinker.EtherCAT_Master_EKxxxx.Beckhoff_EKx9xx.Beckhoff_EKx9xxEK1122.A_0007_EK1960_2608_0019.Module_2_FSOUT.Outputs.Module_2_Channel_2_Standard_Output_X5_6 <-> Module 2 (FSOUT)/Outputs/Module 2.Channel 2.Standard Output (X5.6)
//     PlcTask Outputs/GVL_iXlinker.EtherCAT_Master_EKxxxx.Beckhoff_EKx9xx.Beckhoff_EKx9xxEK1122.A_0007_EK1960_2608_0019.Module_2_FSOUT.Outputs.Module_2_Channel_3_Standard_Output_X5_7 <-> Module 2 (FSOUT)/Outputs/Module 2.Channel 3.Standard Output (X5.7)
//     PlcTask Outputs/GVL_iXlinker.EtherCAT_Master_EKxxxx.Beckhoff_EKx9xx.Beckhoff_EKx9xxEK1122.A_0007_EK1960_2608_0019.Module_2_FSOUT.Outputs.Module_2_Channel_4_Standard_Output_X5_8 <-> Module 2 (FSOUT)/Outputs/Module 2.Channel 4.Standard Output (X5.8)
//     PlcTask Outputs/GVL_iXlinker.EtherCAT_Master_EKxxxx.Beckhoff_EKx9xx.Beckhoff_EKx9xxEK1122.A_0007_EK1960_2608_0019.Module_2_FSOUT.Outputs.Module_3_Channel_1_Standard_Output_X7_1 <-> Module 2 (FSOUT)/Outputs/Module 3.Channel 1.Standard Output (X7.1)
//     PlcTask Outputs/GVL_iXlinker.EtherCAT_Master_EKxxxx.Beckhoff_EKx9xx.Beckhoff_EKx9xxEK1122.A_0007_EK1960_2608_0019.Module_2_FSOUT.Outputs.Module_3_Channel_2_Standard_Output_X7_2 <-> Module 2 (FSOUT)/Outputs/Module 3.Channel 2.Standard Output (X7.2)
//     PlcTask Outputs/GVL_iXlinker.EtherCAT_Master_EKxxxx.Beckhoff_EKx9xx.Beckhoff_EKx9xxEK1122.A_0007_EK1960_2608_0019.Module_2_FSOUT.Outputs.Module_3_Channel_3_Standard_Output_X7_3 <-> Module 2 (FSOUT)/Outputs/Module 3.Channel 3.Standard Output (X7.3)
//     PlcTask Outputs/GVL_iXlinker.EtherCAT_Master_EKxxxx.Beckhoff_EKx9xx.Beckhoff_EKx9xxEK1122.A_0007_EK1960_2608_0019.Module_2_FSOUT.Outputs.Module_3_Channel_4_Standard_Output_X7_4 <-> Module 2 (FSOUT)/Outputs/Module 3.Channel 4.Standard Output (X7.4)
//     PlcTask Outputs/GVL_iXlinker.EtherCAT_Master_EKxxxx.Beckhoff_EKx9xx.Beckhoff_EKx9xxEK1122.A_0007_EK1960_2608_0019.Module_2_FSOUT.Outputs.Module_4_Channel_1_Standard_Output_X7_5 <-> Module 2 (FSOUT)/Outputs/Module 4.Channel 1.Standard Output (X7.5)
//     PlcTask Outputs/GVL_iXlinker.EtherCAT_Master_EKxxxx.Beckhoff_EKx9xx.Beckhoff_EKx9xxEK1122.A_0007_EK1960_2608_0019.Module_2_FSOUT.Outputs.Module_4_Channel_2_Standard_Output_X7_6 <-> Module 2 (FSOUT)/Outputs/Module 4.Channel 2.Standard Output (X7.6)
//     PlcTask Outputs/GVL_iXlinker.EtherCAT_Master_EKxxxx.Beckhoff_EKx9xx.Beckhoff_EKx9xxEK1122.A_0007_EK1960_2608_0019.Module_2_FSOUT.Outputs.Module_4_Channel_3_Standard_Output_X7_7 <-> Module 2 (FSOUT)/Outputs/Module 4.Channel 3.Standard Output (X7.7)
//     PlcTask Outputs/GVL_iXlinker.EtherCAT_Master_EKxxxx.Beckhoff_EKx9xx.Beckhoff_EKx9xxEK1122.A_0007_EK1960_2608_0019.Module_2_FSOUT.Outputs.Module_4_Channel_4_Standard_Output_X7_8 <-> Module 2 (FSOUT)/Outputs/Module 4.Channel 4.Standard Output (X7.8)
//     PlcTask Outputs/GVL_iXlinker.EtherCAT_Master_EKxxxx.Beckhoff_EKx9xx.Beckhoff_EKx9xxEK1122.A_0007_EK1960_2608_0019.Module_2_FSOUT.Outputs.Module_5_Channel_1_Standard_Output_X9_1 <-> Module 2 (FSOUT)/Outputs/Module 5.Channel 1.Standard Output (X9.1)
//     PlcTask Outputs/GVL_iXlinker.EtherCAT_Master_EKxxxx.Beckhoff_EKx9xx.Beckhoff_EKx9xxEK1122.A_0007_EK1960_2608_0019.Module_2_FSOUT.Outputs.Module_5_Channel_2_Standard_Output_X9_2 <-> Module 2 (FSOUT)/Outputs/Module 5.Channel 2.Standard Output (X9.2)
//     PlcTask Outputs/GVL_iXlinker.EtherCAT_Master_EKxxxx.Beckhoff_EKx9xx.Beckhoff_EKx9xxEK1122.A_0007_EK1960_2608_0019.Module_2_FSOUT.Outputs.Module_5_Channel_3_Standard_Output_X9_3 <-> Module 2 (FSOUT)/Outputs/Module 5.Channel 3.Standard Output (X9.3)
//     PlcTask Outputs/GVL_iXlinker.EtherCAT_Master_EKxxxx.Beckhoff_EKx9xx.Beckhoff_EKx9xxEK1122.A_0007_EK1960_2608_0019.Module_2_FSOUT.Outputs.Module_5_Channel_4_Standard_Output_X9_4 <-> Module 2 (FSOUT)/Outputs/Module 5.Channel 4.Standard Output (X9.4)
//     PlcTask Outputs/GVL_iXlinker.EtherCAT_Master_EKxxxx.Beckhoff_EKx9xx.Beckhoff_EKx9xxEK1122.A_0007_EK1960_2608_0019.Module_2_FSOUT.Outputs.Module_6_Channel_1_Standard_Output_X9_5 <-> Module 2 (FSOUT)/Outputs/Module 6.Channel 1.Standard Output (X9.5)
//     PlcTask Outputs/GVL_iXlinker.EtherCAT_Master_EKxxxx.Beckhoff_EKx9xx.Beckhoff_EKx9xxEK1122.A_0007_EK1960_2608_0019.Module_2_FSOUT.Outputs.Module_6_Channel_2_Standard_Output_X9_6 <-> Module 2 (FSOUT)/Outputs/Module 6.Channel 2.Standard Output (X9.6)
//     PlcTask Outputs/GVL_iXlinker.EtherCAT_Master_EKxxxx.Beckhoff_EKx9xx.Beckhoff_EKx9xxEK1122.A_0007_EK1960_2608_0019.Module_2_FSOUT.Outputs.Module_6_Channel_3_Standard_Output_X9_7 <-> Module 2 (FSOUT)/Outputs/Module 6.Channel 3.Standard Output (X9.7)
//     PlcTask Outputs/GVL_iXlinker.EtherCAT_Master_EKxxxx.Beckhoff_EKx9xx.Beckhoff_EKx9xxEK1122.A_0007_EK1960_2608_0019.Module_2_FSOUT.Outputs.Module_6_Channel_4_Standard_Output_X9_8 <-> Module 2 (FSOUT)/Outputs/Module 6.Channel 4.Standard Output (X9.8)
//     PlcTask Outputs/GVL_iXlinker.EtherCAT_Master_EKxxxx.Beckhoff_EKx9xx.Beckhoff_EKx9xxEK1122.A_0007_EK1960_2608_0019.Module_2_FSOUT.Outputs.Relais_Module_Channel_1_Standard_Output_X4_1_X4_5 <-> Module 2 (FSOUT)/Outputs/Relais Module.Channel 1.Standard Output (X4.1, X4.5)
//     PlcTask Outputs/GVL_iXlinker.EtherCAT_Master_EKxxxx.Beckhoff_EKx9xx.Beckhoff_EKx9xxEK1122.A_0007_EK1960_2608_0019.Module_2_FSOUT.Outputs.Relais_Module_Channel_2_Standard_Output_X4_2_X4_6 <-> Module 2 (FSOUT)/Outputs/Relais Module.Channel 2.Standard Output (X4.2, X4.6)
//     PlcTask Outputs/GVL_iXlinker.EtherCAT_Master_EKxxxx.Beckhoff_EKx9xx.Beckhoff_EKx9xxEK1122.A_0007_EK1960_2608_0019.Module_2_FSOUT.Outputs.Relais_Module_Channel_3_Standard_Output_X4_3_X4_7 <-> Module 2 (FSOUT)/Outputs/Relais Module.Channel 3.Standard Output (X4.3, X4.7)
//     PlcTask Outputs/GVL_iXlinker.EtherCAT_Master_EKxxxx.Beckhoff_EKx9xx.Beckhoff_EKx9xxEK1122.A_0007_EK1960_2608_0019.Module_2_FSOUT.Outputs.Relais_Module_Channel_4_Standard_Output_X4_4_X4_8 <-> Module 2 (FSOUT)/Outputs/Relais Module.Channel 4.Standard Output (X4.4, X4.8)
//     PlcTask Inputs/GVL_iXlinker.EtherCAT_Master_EKxxxx.Beckhoff_EKx9xx.Beckhoff_EKx9xxEK1122.A_0007_EK1960_2608_0019.Module_3_FSLOGIC.FSLOGIC_Inputs.Safe_Logic_State <-> Module 3 (FSLOGIC)/FSLOGIC Inputs/Safe Logic State
//     PlcTask Inputs/GVL_iXlinker.EtherCAT_Master_EKxxxx.Beckhoff_EKx9xx.Beckhoff_EKx9xxEK1122.A_0007_EK1960_2608_0019.Module_3_FSLOGIC.FSLOGIC_Inputs.Cycle_Counter <-> Module 3 (FSLOGIC)/FSLOGIC Inputs/Cycle Counter
//     PlcTask Inputs/GVL_iXlinker.EtherCAT_Master_EKxxxx.Beckhoff_EKx9xx.Beckhoff_EKx9xxEK1122.A_0007_EK1960_2608_0019.WcState.WcState0 <-> WcState/WcState0
//     PlcTask Inputs/GVL_iXlinker.EtherCAT_Master_EKxxxx.Beckhoff_EKx9xx.Beckhoff_EKx9xxEK1122.A_0007_EK1960_2608_0019.WcState.WcState1 <-> WcState/WcState1
//     PlcTask Inputs/GVL_iXlinker.EtherCAT_Master_EKxxxx.Beckhoff_EKx9xx.Beckhoff_EKx9xxEK1122.A_0007_EK1960_2608_0019.WcState.InputToggle0 <-> WcState/InputToggle0
//     PlcTask Inputs/GVL_iXlinker.EtherCAT_Master_EKxxxx.Beckhoff_EKx9xx.Beckhoff_EKx9xxEK1122.A_0007_EK1960_2608_0019.WcState.InputToggle1 <-> WcState/InputToggle1
//     PlcTask Inputs/GVL_iXlinker.EtherCAT_Master_EKxxxx.Beckhoff_EKx9xx.Beckhoff_EKx9xxEK1122.A_0007_EK1960_2608_0019.InfoData.AdsAddr <-> InfoData/AdsAddr
//     PlcTask Inputs/GVL_iXlinker.EtherCAT_Master_EKxxxx.Beckhoff_EKx9xx.Beckhoff_EKx9xxEK1122.A_0007_EK1960_2608_0019.InfoData.State <-> InfoData/State
//   PLC/PLC Instance <-> EtherCAT Master EKxxxx/Beckhoff EKx9xx/Beckhoff EKx9xxEK1122/A_0008(EK1960-2608-0021)
//     PlcTask Inputs/GVL_iXlinker.EtherCAT_Master_EKxxxx.Beckhoff_EKx9xx.Beckhoff_EKx9xxEK1122.A_0008_EK1960_2608_0021.Module_1_FSoE.FSoE_Inputs.FSOE/FSoE_Command <-> Module 1 (FSoE)/FSoE Inputs/FSOE/FSoE Command
//     PlcTask Inputs/GVL_iXlinker.EtherCAT_Master_EKxxxx.Beckhoff_EKx9xx.Beckhoff_EKx9xxEK1122.A_0008_EK1960_2608_0021.Module_1_FSoE.FSoE_Inputs.FSOE/FSOUT_Module_1_Module_Fault <-> Module 1 (FSoE)/FSoE Inputs/FSOE/FSOUT Module 1.Module Fault
//     PlcTask Inputs/GVL_iXlinker.EtherCAT_Master_EKxxxx.Beckhoff_EKx9xx.Beckhoff_EKx9xxEK1122.A_0008_EK1960_2608_0021.Module_1_FSoE.FSoE_Inputs.FSOE/FSOUT_Module_2_Module_Fault <-> Module 1 (FSoE)/FSoE Inputs/FSOE/FSOUT Module 2.Module Fault
//     PlcTask Inputs/GVL_iXlinker.EtherCAT_Master_EKxxxx.Beckhoff_EKx9xx.Beckhoff_EKx9xxEK1122.A_0008_EK1960_2608_0021.Module_1_FSoE.FSoE_Inputs.FSOE/FSOUT_Module_3_Module_Fault <-> Module 1 (FSoE)/FSoE Inputs/FSOE/FSOUT Module 3.Module Fault
//     PlcTask Inputs/GVL_iXlinker.EtherCAT_Master_EKxxxx.Beckhoff_EKx9xx.Beckhoff_EKx9xxEK1122.A_0008_EK1960_2608_0021.Module_1_FSoE.FSoE_Inputs.FSOE/FSOUT_Module_4_Module_Fault <-> Module 1 (FSoE)/FSoE Inputs/FSOE/FSOUT Module 4.Module Fault
//     PlcTask Inputs/GVL_iXlinker.EtherCAT_Master_EKxxxx.Beckhoff_EKx9xx.Beckhoff_EKx9xxEK1122.A_0008_EK1960_2608_0021.Module_1_FSoE.FSoE_Inputs.FSOE/FSOUT_Module_5_Module_Fault <-> Module 1 (FSoE)/FSoE Inputs/FSOE/FSOUT Module 5.Module Fault
//     PlcTask Inputs/GVL_iXlinker.EtherCAT_Master_EKxxxx.Beckhoff_EKx9xx.Beckhoff_EKx9xxEK1122.A_0008_EK1960_2608_0021.Module_1_FSoE.FSoE_Inputs.FSOE/FSOUT_Module_6_Module_Fault <-> Module 1 (FSoE)/FSoE Inputs/FSOE/FSOUT Module 6.Module Fault
//     PlcTask Inputs/GVL_iXlinker.EtherCAT_Master_EKxxxx.Beckhoff_EKx9xx.Beckhoff_EKx9xxEK1122.A_0008_EK1960_2608_0021.Module_1_FSoE.FSoE_Inputs.FSOE/FSOUT_Relais_Module_Module_Fault <-> Module 1 (FSoE)/FSoE Inputs/FSOE/FSOUT Relais Module.Module Fault
//     PlcTask Inputs/GVL_iXlinker.EtherCAT_Master_EKxxxx.Beckhoff_EKx9xx.Beckhoff_EKx9xxEK1122.A_0008_EK1960_2608_0021.Module_1_FSoE.FSoE_Inputs.FSOE/FSIN_Module_1_Channel_1_Input_X6_1 <-> Module 1 (FSoE)/FSoE Inputs/FSOE/FSIN Module 1.Channel 1.Input (X6.1)
//     PlcTask Inputs/GVL_iXlinker.EtherCAT_Master_EKxxxx.Beckhoff_EKx9xx.Beckhoff_EKx9xxEK1122.A_0008_EK1960_2608_0021.Module_1_FSoE.FSoE_Inputs.FSOE/FSIN_Module_1_Channel_2_Input_X6_2 <-> Module 1 (FSoE)/FSoE Inputs/FSOE/FSIN Module 1.Channel 2.Input (X6.2)
//     PlcTask Inputs/GVL_iXlinker.EtherCAT_Master_EKxxxx.Beckhoff_EKx9xx.Beckhoff_EKx9xxEK1122.A_0008_EK1960_2608_0021.Module_1_FSoE.FSoE_Inputs.FSOE/FSIN_Module_2_Channel_1_Input_X6_3 <-> Module 1 (FSoE)/FSoE Inputs/FSOE/FSIN Module 2.Channel 1.Input (X6.3)
//     PlcTask Inputs/GVL_iXlinker.EtherCAT_Master_EKxxxx.Beckhoff_EKx9xx.Beckhoff_EKx9xxEK1122.A_0008_EK1960_2608_0021.Module_1_FSoE.FSoE_Inputs.FSOE/FSIN_Module_2_Channel_2_Input_X6_4 <-> Module 1 (FSoE)/FSoE Inputs/FSOE/FSIN Module 2.Channel 2.Input (X6.4)
//     PlcTask Inputs/GVL_iXlinker.EtherCAT_Master_EKxxxx.Beckhoff_EKx9xx.Beckhoff_EKx9xxEK1122.A_0008_EK1960_2608_0021.Module_1_FSoE.FSoE_Inputs.FSOE/FSIN_Module_3_Channel_1_Input_X6_5 <-> Module 1 (FSoE)/FSoE Inputs/FSOE/FSIN Module 3.Channel 1.Input (X6.5)
//     PlcTask Inputs/GVL_iXlinker.EtherCAT_Master_EKxxxx.Beckhoff_EKx9xx.Beckhoff_EKx9xxEK1122.A_0008_EK1960_2608_0021.Module_1_FSoE.FSoE_Inputs.FSOE/FSIN_Module_3_Channel_2_Input_X6_6 <-> Module 1 (FSoE)/FSoE Inputs/FSOE/FSIN Module 3.Channel 2.Input (X6.6)
//     PlcTask Inputs/GVL_iXlinker.EtherCAT_Master_EKxxxx.Beckhoff_EKx9xx.Beckhoff_EKx9xxEK1122.A_0008_EK1960_2608_0021.Module_1_FSoE.FSoE_Inputs.FSOE/FSIN_Module_4_Channel_1_Input_X6_7 <-> Module 1 (FSoE)/FSoE Inputs/FSOE/FSIN Module 4.Channel 1.Input (X6.7)
//     PlcTask Inputs/GVL_iXlinker.EtherCAT_Master_EKxxxx.Beckhoff_EKx9xx.Beckhoff_EKx9xxEK1122.A_0008_EK1960_2608_0021.Module_1_FSoE.FSoE_Inputs.FSOE/FSIN_Module_4_Channel_2_Input_X6_8 <-> Module 1 (FSoE)/FSoE Inputs/FSOE/FSIN Module 4.Channel 2.Input (X6.8)
//     PlcTask Inputs/GVL_iXlinker.EtherCAT_Master_EKxxxx.Beckhoff_EKx9xx.Beckhoff_EKx9xxEK1122.A_0008_EK1960_2608_0021.Module_1_FSoE.FSoE_Inputs.FSOE/FSIN_Module_5_Channel_1_Input_X6_9 <-> Module 1 (FSoE)/FSoE Inputs/FSOE/FSIN Module 5.Channel 1.Input (X6.9)
//     PlcTask Inputs/GVL_iXlinker.EtherCAT_Master_EKxxxx.Beckhoff_EKx9xx.Beckhoff_EKx9xxEK1122.A_0008_EK1960_2608_0021.Module_1_FSoE.FSoE_Inputs.FSOE/FSIN_Module_5_Channel_2_Input_X6_10 <-> Module 1 (FSoE)/FSoE Inputs/FSOE/FSIN Module 5.Channel 2.Input (X6.10)
//     PlcTask Inputs/GVL_iXlinker.EtherCAT_Master_EKxxxx.Beckhoff_EKx9xx.Beckhoff_EKx9xxEK1122.A_0008_EK1960_2608_0021.Module_1_FSoE.FSoE_Inputs.FSOE/FSIN_Module_6_Channel_1_Input_X8_1 <-> Module 1 (FSoE)/FSoE Inputs/FSOE/FSIN Module 6.Channel 1.Input (X8.1)
//     PlcTask Inputs/GVL_iXlinker.EtherCAT_Master_EKxxxx.Beckhoff_EKx9xx.Beckhoff_EKx9xxEK1122.A_0008_EK1960_2608_0021.Module_1_FSoE.FSoE_Inputs.FSOE/FSIN_Module_6_Channel_2_Input_X8_2 <-> Module 1 (FSoE)/FSoE Inputs/FSOE/FSIN Module 6.Channel 2.Input (X8.2)
//     PlcTask Inputs/GVL_iXlinker.EtherCAT_Master_EKxxxx.Beckhoff_EKx9xx.Beckhoff_EKx9xxEK1122.A_0008_EK1960_2608_0021.Module_1_FSoE.FSoE_Inputs.FSOE/FSIN_Module_7_Channel_1_Input_X8_3 <-> Module 1 (FSoE)/FSoE Inputs/FSOE/FSIN Module 7.Channel 1.Input (X8.3)
//     PlcTask Inputs/GVL_iXlinker.EtherCAT_Master_EKxxxx.Beckhoff_EKx9xx.Beckhoff_EKx9xxEK1122.A_0008_EK1960_2608_0021.Module_1_FSoE.FSoE_Inputs.FSOE/FSIN_Module_7_Channel_2_Input_X8_4 <-> Module 1 (FSoE)/FSoE Inputs/FSOE/FSIN Module 7.Channel 2.Input (X8.4)
//     PlcTask Inputs/GVL_iXlinker.EtherCAT_Master_EKxxxx.Beckhoff_EKx9xx.Beckhoff_EKx9xxEK1122.A_0008_EK1960_2608_0021.Module_1_FSoE.FSoE_Inputs.FSOE/FSIN_Module_8_Channel_1_Input_X8_5 <-> Module 1 (FSoE)/FSoE Inputs/FSOE/FSIN Module 8.Channel 1.Input (X8.5)
//     PlcTask Inputs/GVL_iXlinker.EtherCAT_Master_EKxxxx.Beckhoff_EKx9xx.Beckhoff_EKx9xxEK1122.A_0008_EK1960_2608_0021.Module_1_FSoE.FSoE_Inputs.FSOE/FSIN_Module_8_Channel_2_Input_X8_6 <-> Module 1 (FSoE)/FSoE Inputs/FSOE/FSIN Module 8.Channel 2.Input (X8.6)
//     PlcTask Inputs/GVL_iXlinker.EtherCAT_Master_EKxxxx.Beckhoff_EKx9xx.Beckhoff_EKx9xxEK1122.A_0008_EK1960_2608_0021.Module_1_FSoE.FSoE_Inputs.FSOE/FSIN_Module_9_Channel_1_Input_X8_7 <-> Module 1 (FSoE)/FSoE Inputs/FSOE/FSIN Module 9.Channel 1.Input (X8.7)
//     PlcTask Inputs/GVL_iXlinker.EtherCAT_Master_EKxxxx.Beckhoff_EKx9xx.Beckhoff_EKx9xxEK1122.A_0008_EK1960_2608_0021.Module_1_FSoE.FSoE_Inputs.FSOE/FSIN_Module_9_Channel_2_Input_X8_8 <-> Module 1 (FSoE)/FSoE Inputs/FSOE/FSIN Module 9.Channel 2.Input (X8.8)
//     PlcTask Inputs/GVL_iXlinker.EtherCAT_Master_EKxxxx.Beckhoff_EKx9xx.Beckhoff_EKx9xxEK1122.A_0008_EK1960_2608_0021.Module_1_FSoE.FSoE_Inputs.FSOE/FSIN_Module_10_Channel_1_Input_X8_9 <-> Module 1 (FSoE)/FSoE Inputs/FSOE/FSIN Module 10.Channel 1.Input (X8.9)
//     PlcTask Inputs/GVL_iXlinker.EtherCAT_Master_EKxxxx.Beckhoff_EKx9xx.Beckhoff_EKx9xxEK1122.A_0008_EK1960_2608_0021.Module_1_FSoE.FSoE_Inputs.FSOE/FSIN_Module_10_Channel_2_Input_X8_10 <-> Module 1 (FSoE)/FSoE Inputs/FSOE/FSIN Module 10.Channel 2.Input (X8.10)
//     PlcTask Inputs/GVL_iXlinker.EtherCAT_Master_EKxxxx.Beckhoff_EKx9xx.Beckhoff_EKx9xxEK1122.A_0008_EK1960_2608_0021.Module_1_FSoE.FSoE_Inputs.FSOE/FSIN_Module_1_Module_Fault <-> Module 1 (FSoE)/FSoE Inputs/FSOE/FSIN Module 1.Module Fault
//     PlcTask Inputs/GVL_iXlinker.EtherCAT_Master_EKxxxx.Beckhoff_EKx9xx.Beckhoff_EKx9xxEK1122.A_0008_EK1960_2608_0021.Module_1_FSoE.FSoE_Inputs.FSOE/FSIN_Module_2_Module_Fault <-> Module 1 (FSoE)/FSoE Inputs/FSOE/FSIN Module 2.Module Fault
//     PlcTask Inputs/GVL_iXlinker.EtherCAT_Master_EKxxxx.Beckhoff_EKx9xx.Beckhoff_EKx9xxEK1122.A_0008_EK1960_2608_0021.Module_1_FSoE.FSoE_Inputs.FSOE/FSIN_Module_3_Module_Fault <-> Module 1 (FSoE)/FSoE Inputs/FSOE/FSIN Module 3.Module Fault
//     PlcTask Inputs/GVL_iXlinker.EtherCAT_Master_EKxxxx.Beckhoff_EKx9xx.Beckhoff_EKx9xxEK1122.A_0008_EK1960_2608_0021.Module_1_FSoE.FSoE_Inputs.FSOE/FSIN_Module_4_Module_Fault <-> Module 1 (FSoE)/FSoE Inputs/FSOE/FSIN Module 4.Module Fault
//     PlcTask Inputs/GVL_iXlinker.EtherCAT_Master_EKxxxx.Beckhoff_EKx9xx.Beckhoff_EKx9xxEK1122.A_0008_EK1960_2608_0021.Module_1_FSoE.FSoE_Inputs.FSOE/FSIN_Module_5_Module_Fault <-> Module 1 (FSoE)/FSoE Inputs/FSOE/FSIN Module 5.Module Fault
//     PlcTask Inputs/GVL_iXlinker.EtherCAT_Master_EKxxxx.Beckhoff_EKx9xx.Beckhoff_EKx9xxEK1122.A_0008_EK1960_2608_0021.Module_1_FSoE.FSoE_Inputs.FSOE/FSIN_Module_6_Module_Fault <-> Module 1 (FSoE)/FSoE Inputs/FSOE/FSIN Module 6.Module Fault
//     PlcTask Inputs/GVL_iXlinker.EtherCAT_Master_EKxxxx.Beckhoff_EKx9xx.Beckhoff_EKx9xxEK1122.A_0008_EK1960_2608_0021.Module_1_FSoE.FSoE_Inputs.FSOE/FSIN_Module_7_Module_Fault <-> Module 1 (FSoE)/FSoE Inputs/FSOE/FSIN Module 7.Module Fault
//     PlcTask Inputs/GVL_iXlinker.EtherCAT_Master_EKxxxx.Beckhoff_EKx9xx.Beckhoff_EKx9xxEK1122.A_0008_EK1960_2608_0021.Module_1_FSoE.FSoE_Inputs.FSOE/FSIN_Module_8_Module_Fault <-> Module 1 (FSoE)/FSoE Inputs/FSOE/FSIN Module 8.Module Fault
//     PlcTask Inputs/GVL_iXlinker.EtherCAT_Master_EKxxxx.Beckhoff_EKx9xx.Beckhoff_EKx9xxEK1122.A_0008_EK1960_2608_0021.Module_1_FSoE.FSoE_Inputs.FSOE/FSoE_CRC_000 <-> Module 1 (FSoE)/FSoE Inputs/FSOE/FSoE CRC 000
//     PlcTask Inputs/GVL_iXlinker.EtherCAT_Master_EKxxxx.Beckhoff_EKx9xx.Beckhoff_EKx9xxEK1122.A_0008_EK1960_2608_0021.Module_1_FSoE.FSoE_Inputs.FSOE/FSoE_CRC_001 <-> Module 1 (FSoE)/FSoE Inputs/FSOE/FSoE CRC 001
//     PlcTask Inputs/GVL_iXlinker.EtherCAT_Master_EKxxxx.Beckhoff_EKx9xx.Beckhoff_EKx9xxEK1122.A_0008_EK1960_2608_0021.Module_1_FSoE.FSoE_Inputs.FSOE/FSoE_CRC_002 <-> Module 1 (FSoE)/FSoE Inputs/FSOE/FSoE CRC 002
//     PlcTask Inputs/GVL_iXlinker.EtherCAT_Master_EKxxxx.Beckhoff_EKx9xx.Beckhoff_EKx9xxEK1122.A_0008_EK1960_2608_0021.Module_1_FSoE.FSoE_Inputs.FSOE/FSIN_Module_9_Module_Fault_1 <-> Module 1 (FSoE)/FSoE Inputs/FSOE/FSIN Module 9.Module Fault 1
//     PlcTask Inputs/GVL_iXlinker.EtherCAT_Master_EKxxxx.Beckhoff_EKx9xx.Beckhoff_EKx9xxEK1122.A_0008_EK1960_2608_0021.Module_1_FSoE.FSoE_Inputs.FSOE/FSIN_Module_9_Module_Fault_2 <-> Module 1 (FSoE)/FSoE Inputs/FSOE/FSIN Module 9.Module Fault 2
//     PlcTask Inputs/GVL_iXlinker.EtherCAT_Master_EKxxxx.Beckhoff_EKx9xx.Beckhoff_EKx9xxEK1122.A_0008_EK1960_2608_0021.Module_1_FSoE.FSoE_Inputs.FSOE/FSIN_Module_10_Module_Fault_1 <-> Module 1 (FSoE)/FSoE Inputs/FSOE/FSIN Module 10.Module Fault 1
//     PlcTask Inputs/GVL_iXlinker.EtherCAT_Master_EKxxxx.Beckhoff_EKx9xx.Beckhoff_EKx9xxEK1122.A_0008_EK1960_2608_0021.Module_1_FSoE.FSoE_Inputs.FSOE/FSIN_Module_10_Module_Fault_2 <-> Module 1 (FSoE)/FSoE Inputs/FSOE/FSIN Module 10.Module Fault 2
//     PlcTask Inputs/GVL_iXlinker.EtherCAT_Master_EKxxxx.Beckhoff_EKx9xx.Beckhoff_EKx9xxEK1122.A_0008_EK1960_2608_0021.Module_1_FSoE.FSoE_Inputs.FSOE/FSoE_Connection_ID <-> Module 1 (FSoE)/FSoE Inputs/FSOE/FSoE Connection ID
//     PlcTask Outputs/GVL_iXlinker.EtherCAT_Master_EKxxxx.Beckhoff_EKx9xx.Beckhoff_EKx9xxEK1122.A_0008_EK1960_2608_0021.Module_1_FSoE.FSoE_Outputs.FSOE/FSoE_Command <-> Module 1 (FSoE)/FSoE Outputs/FSOE/FSoE Command
//     PlcTask Outputs/GVL_iXlinker.EtherCAT_Master_EKxxxx.Beckhoff_EKx9xx.Beckhoff_EKx9xxEK1122.A_0008_EK1960_2608_0021.Module_1_FSoE.FSoE_Outputs.FSOE/FSOUT_Module_1_Channel_1_Output_X5_1 <-> Module 1 (FSoE)/FSoE Outputs/FSOE/FSOUT Module 1.Channel 1.Output (X5.1)
//     PlcTask Outputs/GVL_iXlinker.EtherCAT_Master_EKxxxx.Beckhoff_EKx9xx.Beckhoff_EKx9xxEK1122.A_0008_EK1960_2608_0021.Module_1_FSoE.FSoE_Outputs.FSOE/FSOUT_Module_1_Channel_2_Output_X5_2 <-> Module 1 (FSoE)/FSoE Outputs/FSOE/FSOUT Module 1.Channel 2.Output (X5.2)
//     PlcTask Outputs/GVL_iXlinker.EtherCAT_Master_EKxxxx.Beckhoff_EKx9xx.Beckhoff_EKx9xxEK1122.A_0008_EK1960_2608_0021.Module_1_FSoE.FSoE_Outputs.FSOE/FSOUT_Module_1_Channel_3_Output_X5_3 <-> Module 1 (FSoE)/FSoE Outputs/FSOE/FSOUT Module 1.Channel 3.Output (X5.3)
//     PlcTask Outputs/GVL_iXlinker.EtherCAT_Master_EKxxxx.Beckhoff_EKx9xx.Beckhoff_EKx9xxEK1122.A_0008_EK1960_2608_0021.Module_1_FSoE.FSoE_Outputs.FSOE/FSOUT_Module_1_Channel_4_Output_X5_4 <-> Module 1 (FSoE)/FSoE Outputs/FSOE/FSOUT Module 1.Channel 4.Output (X5.4)
//     PlcTask Outputs/GVL_iXlinker.EtherCAT_Master_EKxxxx.Beckhoff_EKx9xx.Beckhoff_EKx9xxEK1122.A_0008_EK1960_2608_0021.Module_1_FSoE.FSoE_Outputs.FSOE/FSOUT_Module_2_Channel_1_Output_X5_5 <-> Module 1 (FSoE)/FSoE Outputs/FSOE/FSOUT Module 2.Channel 1.Output (X5.5)
//     PlcTask Outputs/GVL_iXlinker.EtherCAT_Master_EKxxxx.Beckhoff_EKx9xx.Beckhoff_EKx9xxEK1122.A_0008_EK1960_2608_0021.Module_1_FSoE.FSoE_Outputs.FSOE/FSOUT_Module_2_Channel_2_Output_X5_6 <-> Module 1 (FSoE)/FSoE Outputs/FSOE/FSOUT Module 2.Channel 2.Output (X5.6)
//     PlcTask Outputs/GVL_iXlinker.EtherCAT_Master_EKxxxx.Beckhoff_EKx9xx.Beckhoff_EKx9xxEK1122.A_0008_EK1960_2608_0021.Module_1_FSoE.FSoE_Outputs.FSOE/FSOUT_Module_2_Channel_3_Output_X5_7 <-> Module 1 (FSoE)/FSoE Outputs/FSOE/FSOUT Module 2.Channel 3.Output (X5.7)
//     PlcTask Outputs/GVL_iXlinker.EtherCAT_Master_EKxxxx.Beckhoff_EKx9xx.Beckhoff_EKx9xxEK1122.A_0008_EK1960_2608_0021.Module_1_FSoE.FSoE_Outputs.FSOE/FSOUT_Module_2_Channel_4_Output_X5_8 <-> Module 1 (FSoE)/FSoE Outputs/FSOE/FSOUT Module 2.Channel 4.Output (X5.8)
//     PlcTask Outputs/GVL_iXlinker.EtherCAT_Master_EKxxxx.Beckhoff_EKx9xx.Beckhoff_EKx9xxEK1122.A_0008_EK1960_2608_0021.Module_1_FSoE.FSoE_Outputs.FSOE/FSOUT_Module_3_Channel_1_Output_X7_1 <-> Module 1 (FSoE)/FSoE Outputs/FSOE/FSOUT Module 3.Channel 1.Output (X7.1)
//     PlcTask Outputs/GVL_iXlinker.EtherCAT_Master_EKxxxx.Beckhoff_EKx9xx.Beckhoff_EKx9xxEK1122.A_0008_EK1960_2608_0021.Module_1_FSoE.FSoE_Outputs.FSOE/FSOUT_Module_3_Channel_2_Output_X7_2 <-> Module 1 (FSoE)/FSoE Outputs/FSOE/FSOUT Module 3.Channel 2.Output (X7.2)
//     PlcTask Outputs/GVL_iXlinker.EtherCAT_Master_EKxxxx.Beckhoff_EKx9xx.Beckhoff_EKx9xxEK1122.A_0008_EK1960_2608_0021.Module_1_FSoE.FSoE_Outputs.FSOE/FSOUT_Module_3_Channel_3_Output_X7_3 <-> Module 1 (FSoE)/FSoE Outputs/FSOE/FSOUT Module 3.Channel 3.Output (X7.3)
//     PlcTask Outputs/GVL_iXlinker.EtherCAT_Master_EKxxxx.Beckhoff_EKx9xx.Beckhoff_EKx9xxEK1122.A_0008_EK1960_2608_0021.Module_1_FSoE.FSoE_Outputs.FSOE/FSOUT_Module_3_Channel_4_Output_X7_4 <-> Module 1 (FSoE)/FSoE Outputs/FSOE/FSOUT Module 3.Channel 4.Output (X7.4)
//     PlcTask Outputs/GVL_iXlinker.EtherCAT_Master_EKxxxx.Beckhoff_EKx9xx.Beckhoff_EKx9xxEK1122.A_0008_EK1960_2608_0021.Module_1_FSoE.FSoE_Outputs.FSOE/FSOUT_Module_4_Channel_1_Output_X7_5 <-> Module 1 (FSoE)/FSoE Outputs/FSOE/FSOUT Module 4.Channel 1.Output (X7.5)
//     PlcTask Outputs/GVL_iXlinker.EtherCAT_Master_EKxxxx.Beckhoff_EKx9xx.Beckhoff_EKx9xxEK1122.A_0008_EK1960_2608_0021.Module_1_FSoE.FSoE_Outputs.FSOE/FSOUT_Module_4_Channel_2_Output_X7_6 <-> Module 1 (FSoE)/FSoE Outputs/FSOE/FSOUT Module 4.Channel 2.Output (X7.6)
//     PlcTask Outputs/GVL_iXlinker.EtherCAT_Master_EKxxxx.Beckhoff_EKx9xx.Beckhoff_EKx9xxEK1122.A_0008_EK1960_2608_0021.Module_1_FSoE.FSoE_Outputs.FSOE/FSOUT_Module_4_Channel_3_Output_X7_7 <-> Module 1 (FSoE)/FSoE Outputs/FSOE/FSOUT Module 4.Channel 3.Output (X7.7)
//     PlcTask Outputs/GVL_iXlinker.EtherCAT_Master_EKxxxx.Beckhoff_EKx9xx.Beckhoff_EKx9xxEK1122.A_0008_EK1960_2608_0021.Module_1_FSoE.FSoE_Outputs.FSOE/FSOUT_Module_4_Channel_4_Output_X7_8 <-> Module 1 (FSoE)/FSoE Outputs/FSOE/FSOUT Module 4.Channel 4.Output (X7.8)
//     PlcTask Outputs/GVL_iXlinker.EtherCAT_Master_EKxxxx.Beckhoff_EKx9xx.Beckhoff_EKx9xxEK1122.A_0008_EK1960_2608_0021.Module_1_FSoE.FSoE_Outputs.FSOE/FSOUT_Module_5_Channel_1_Output_X9_1 <-> Module 1 (FSoE)/FSoE Outputs/FSOE/FSOUT Module 5.Channel 1.Output (X9.1)
//     PlcTask Outputs/GVL_iXlinker.EtherCAT_Master_EKxxxx.Beckhoff_EKx9xx.Beckhoff_EKx9xxEK1122.A_0008_EK1960_2608_0021.Module_1_FSoE.FSoE_Outputs.FSOE/FSOUT_Module_5_Channel_2_Output_X9_2 <-> Module 1 (FSoE)/FSoE Outputs/FSOE/FSOUT Module 5.Channel 2.Output (X9.2)
//     PlcTask Outputs/GVL_iXlinker.EtherCAT_Master_EKxxxx.Beckhoff_EKx9xx.Beckhoff_EKx9xxEK1122.A_0008_EK1960_2608_0021.Module_1_FSoE.FSoE_Outputs.FSOE/FSOUT_Module_5_Channel_3_Output_X9_3 <-> Module 1 (FSoE)/FSoE Outputs/FSOE/FSOUT Module 5.Channel 3.Output (X9.3)
//     PlcTask Outputs/GVL_iXlinker.EtherCAT_Master_EKxxxx.Beckhoff_EKx9xx.Beckhoff_EKx9xxEK1122.A_0008_EK1960_2608_0021.Module_1_FSoE.FSoE_Outputs.FSOE/FSOUT_Module_5_Channel_4_Output_X9_4 <-> Module 1 (FSoE)/FSoE Outputs/FSOE/FSOUT Module 5.Channel 4.Output (X9.4)
//     PlcTask Outputs/GVL_iXlinker.EtherCAT_Master_EKxxxx.Beckhoff_EKx9xx.Beckhoff_EKx9xxEK1122.A_0008_EK1960_2608_0021.Module_1_FSoE.FSoE_Outputs.FSOE/FSOUT_Module_6_Channel_1_Output_X9_5 <-> Module 1 (FSoE)/FSoE Outputs/FSOE/FSOUT Module 6.Channel 1.Output (X9.5)
//     PlcTask Outputs/GVL_iXlinker.EtherCAT_Master_EKxxxx.Beckhoff_EKx9xx.Beckhoff_EKx9xxEK1122.A_0008_EK1960_2608_0021.Module_1_FSoE.FSoE_Outputs.FSOE/FSOUT_Module_6_Channel_2_Output_X9_6 <-> Module 1 (FSoE)/FSoE Outputs/FSOE/FSOUT Module 6.Channel 2.Output (X9.6)
//     PlcTask Outputs/GVL_iXlinker.EtherCAT_Master_EKxxxx.Beckhoff_EKx9xx.Beckhoff_EKx9xxEK1122.A_0008_EK1960_2608_0021.Module_1_FSoE.FSoE_Outputs.FSOE/FSOUT_Module_6_Channel_3_Output_X9_7 <-> Module 1 (FSoE)/FSoE Outputs/FSOE/FSOUT Module 6.Channel 3.Output (X9.7)
//     PlcTask Outputs/GVL_iXlinker.EtherCAT_Master_EKxxxx.Beckhoff_EKx9xx.Beckhoff_EKx9xxEK1122.A_0008_EK1960_2608_0021.Module_1_FSoE.FSoE_Outputs.FSOE/FSOUT_Module_6_Channel_4_Output_X9_8 <-> Module 1 (FSoE)/FSoE Outputs/FSOE/FSOUT Module 6.Channel 4.Output (X9.8)
//     PlcTask Outputs/GVL_iXlinker.EtherCAT_Master_EKxxxx.Beckhoff_EKx9xx.Beckhoff_EKx9xxEK1122.A_0008_EK1960_2608_0021.Module_1_FSoE.FSoE_Outputs.FSOE/FSOUT_Module_1_ErrAck <-> Module 1 (FSoE)/FSoE Outputs/FSOE/FSOUT Module 1.ErrAck
//     PlcTask Outputs/GVL_iXlinker.EtherCAT_Master_EKxxxx.Beckhoff_EKx9xx.Beckhoff_EKx9xxEK1122.A_0008_EK1960_2608_0021.Module_1_FSoE.FSoE_Outputs.FSOE/FSOUT_Module_2_ErrAck <-> Module 1 (FSoE)/FSoE Outputs/FSOE/FSOUT Module 2.ErrAck
//     PlcTask Outputs/GVL_iXlinker.EtherCAT_Master_EKxxxx.Beckhoff_EKx9xx.Beckhoff_EKx9xxEK1122.A_0008_EK1960_2608_0021.Module_1_FSoE.FSoE_Outputs.FSOE/FSOUT_Module_3_ErrAck <-> Module 1 (FSoE)/FSoE Outputs/FSOE/FSOUT Module 3.ErrAck
//     PlcTask Outputs/GVL_iXlinker.EtherCAT_Master_EKxxxx.Beckhoff_EKx9xx.Beckhoff_EKx9xxEK1122.A_0008_EK1960_2608_0021.Module_1_FSoE.FSoE_Outputs.FSOE/FSOUT_Module_4_ErrAck <-> Module 1 (FSoE)/FSoE Outputs/FSOE/FSOUT Module 4.ErrAck
//     PlcTask Outputs/GVL_iXlinker.EtherCAT_Master_EKxxxx.Beckhoff_EKx9xx.Beckhoff_EKx9xxEK1122.A_0008_EK1960_2608_0021.Module_1_FSoE.FSoE_Outputs.FSOE/FSOUT_Module_5_ErrAck <-> Module 1 (FSoE)/FSoE Outputs/FSOE/FSOUT Module 5.ErrAck
//     PlcTask Outputs/GVL_iXlinker.EtherCAT_Master_EKxxxx.Beckhoff_EKx9xx.Beckhoff_EKx9xxEK1122.A_0008_EK1960_2608_0021.Module_1_FSoE.FSoE_Outputs.FSOE/FSOUT_Module_6_ErrAck <-> Module 1 (FSoE)/FSoE Outputs/FSOE/FSOUT Module 6.ErrAck
//     PlcTask Outputs/GVL_iXlinker.EtherCAT_Master_EKxxxx.Beckhoff_EKx9xx.Beckhoff_EKx9xxEK1122.A_0008_EK1960_2608_0021.Module_1_FSoE.FSoE_Outputs.FSOE/FSoE_CRC_000 <-> Module 1 (FSoE)/FSoE Outputs/FSOE/FSoE CRC 000
//     PlcTask Outputs/GVL_iXlinker.EtherCAT_Master_EKxxxx.Beckhoff_EKx9xx.Beckhoff_EKx9xxEK1122.A_0008_EK1960_2608_0021.Module_1_FSoE.FSoE_Outputs.FSOE/FSoE_CRC_001 <-> Module 1 (FSoE)/FSoE Outputs/FSOE/FSoE CRC 001
//     PlcTask Outputs/GVL_iXlinker.EtherCAT_Master_EKxxxx.Beckhoff_EKx9xx.Beckhoff_EKx9xxEK1122.A_0008_EK1960_2608_0021.Module_1_FSoE.FSoE_Outputs.FSOE/FSoE_CRC_002 <-> Module 1 (FSoE)/FSoE Outputs/FSOE/FSoE CRC 002
//     PlcTask Outputs/GVL_iXlinker.EtherCAT_Master_EKxxxx.Beckhoff_EKx9xx.Beckhoff_EKx9xxEK1122.A_0008_EK1960_2608_0021.Module_1_FSoE.FSoE_Outputs.FSOE/FSOUT_Relais_Module_Channel_1_Output_X4_1_X4_5 <-> Module 1 (FSoE)/FSoE Outputs/FSOE/FSOUT Relais Module.Channel 1.Output (X4.1, X4.5)
//     PlcTask Outputs/GVL_iXlinker.EtherCAT_Master_EKxxxx.Beckhoff_EKx9xx.Beckhoff_EKx9xxEK1122.A_0008_EK1960_2608_0021.Module_1_FSoE.FSoE_Outputs.FSOE/FSOUT_Relais_Module_Channel_2_Output_X4_2_X4_6 <-> Module 1 (FSoE)/FSoE Outputs/FSOE/FSOUT Relais Module.Channel 2.Output (X4.2, X4.6)
//     PlcTask Outputs/GVL_iXlinker.EtherCAT_Master_EKxxxx.Beckhoff_EKx9xx.Beckhoff_EKx9xxEK1122.A_0008_EK1960_2608_0021.Module_1_FSoE.FSoE_Outputs.FSOE/FSOUT_Relais_Module_Channel_3_Output_X4_3_X4_7 <-> Module 1 (FSoE)/FSoE Outputs/FSOE/FSOUT Relais Module.Channel 3.Output (X4.3, X4.7)
//     PlcTask Outputs/GVL_iXlinker.EtherCAT_Master_EKxxxx.Beckhoff_EKx9xx.Beckhoff_EKx9xxEK1122.A_0008_EK1960_2608_0021.Module_1_FSoE.FSoE_Outputs.FSOE/FSOUT_Relais_Module_Channel_4_Output_X4_4_X4_8 <-> Module 1 (FSoE)/FSoE Outputs/FSOE/FSOUT Relais Module.Channel 4.Output (X4.4, X4.8)
//     PlcTask Outputs/GVL_iXlinker.EtherCAT_Master_EKxxxx.Beckhoff_EKx9xx.Beckhoff_EKx9xxEK1122.A_0008_EK1960_2608_0021.Module_1_FSoE.FSoE_Outputs.FSOE/FSOUT_Relais_Module_ErrAck <-> Module 1 (FSoE)/FSoE Outputs/FSOE/FSOUT Relais Module.ErrAck
//     PlcTask Outputs/GVL_iXlinker.EtherCAT_Master_EKxxxx.Beckhoff_EKx9xx.Beckhoff_EKx9xxEK1122.A_0008_EK1960_2608_0021.Module_1_FSoE.FSoE_Outputs.FSOE/FSIN_Module_1_ErrAck <-> Module 1 (FSoE)/FSoE Outputs/FSOE/FSIN Module 1.ErrAck
//     PlcTask Outputs/GVL_iXlinker.EtherCAT_Master_EKxxxx.Beckhoff_EKx9xx.Beckhoff_EKx9xxEK1122.A_0008_EK1960_2608_0021.Module_1_FSoE.FSoE_Outputs.FSOE/FSIN_Module_2_ErrAck <-> Module 1 (FSoE)/FSoE Outputs/FSOE/FSIN Module 2.ErrAck
//     PlcTask Outputs/GVL_iXlinker.EtherCAT_Master_EKxxxx.Beckhoff_EKx9xx.Beckhoff_EKx9xxEK1122.A_0008_EK1960_2608_0021.Module_1_FSoE.FSoE_Outputs.FSOE/FSIN_Module_3_ErrAck <-> Module 1 (FSoE)/FSoE Outputs/FSOE/FSIN Module 3.ErrAck
//     PlcTask Outputs/GVL_iXlinker.EtherCAT_Master_EKxxxx.Beckhoff_EKx9xx.Beckhoff_EKx9xxEK1122.A_0008_EK1960_2608_0021.Module_1_FSoE.FSoE_Outputs.FSOE/FSIN_Module_4_ErrAck <-> Module 1 (FSoE)/FSoE Outputs/FSOE/FSIN Module 4.ErrAck
//     PlcTask Outputs/GVL_iXlinker.EtherCAT_Master_EKxxxx.Beckhoff_EKx9xx.Beckhoff_EKx9xxEK1122.A_0008_EK1960_2608_0021.Module_1_FSoE.FSoE_Outputs.FSOE/FSIN_Module_5_ErrAck <-> Module 1 (FSoE)/FSoE Outputs/FSOE/FSIN Module 5.ErrAck
//     PlcTask Outputs/GVL_iXlinker.EtherCAT_Master_EKxxxx.Beckhoff_EKx9xx.Beckhoff_EKx9xxEK1122.A_0008_EK1960_2608_0021.Module_1_FSoE.FSoE_Outputs.FSOE/FSIN_Module_6_ErrAck <-> Module 1 (FSoE)/FSoE Outputs/FSOE/FSIN Module 6.ErrAck
//     PlcTask Outputs/GVL_iXlinker.EtherCAT_Master_EKxxxx.Beckhoff_EKx9xx.Beckhoff_EKx9xxEK1122.A_0008_EK1960_2608_0021.Module_1_FSoE.FSoE_Outputs.FSOE/FSIN_Module_7_ErrAck <-> Module 1 (FSoE)/FSoE Outputs/FSOE/FSIN Module 7.ErrAck
//     PlcTask Outputs/GVL_iXlinker.EtherCAT_Master_EKxxxx.Beckhoff_EKx9xx.Beckhoff_EKx9xxEK1122.A_0008_EK1960_2608_0021.Module_1_FSoE.FSoE_Outputs.FSOE/FSIN_Module_8_ErrAck <-> Module 1 (FSoE)/FSoE Outputs/FSOE/FSIN Module 8.ErrAck
//     PlcTask Outputs/GVL_iXlinker.EtherCAT_Master_EKxxxx.Beckhoff_EKx9xx.Beckhoff_EKx9xxEK1122.A_0008_EK1960_2608_0021.Module_1_FSoE.FSoE_Outputs.FSOE/FSIN_Module_9_Err_Ack_1 <-> Module 1 (FSoE)/FSoE Outputs/FSOE/FSIN Module 9.Err Ack 1
//     PlcTask Outputs/GVL_iXlinker.EtherCAT_Master_EKxxxx.Beckhoff_EKx9xx.Beckhoff_EKx9xxEK1122.A_0008_EK1960_2608_0021.Module_1_FSoE.FSoE_Outputs.FSOE/FSIN_Module_9_Err_Ack_2 <-> Module 1 (FSoE)/FSoE Outputs/FSOE/FSIN Module 9.Err Ack 2
//     PlcTask Outputs/GVL_iXlinker.EtherCAT_Master_EKxxxx.Beckhoff_EKx9xx.Beckhoff_EKx9xxEK1122.A_0008_EK1960_2608_0021.Module_1_FSoE.FSoE_Outputs.FSOE/FSIN_Module_10_Err_Ack_1 <-> Module 1 (FSoE)/FSoE Outputs/FSOE/FSIN Module 10.Err Ack 1
//     PlcTask Outputs/GVL_iXlinker.EtherCAT_Master_EKxxxx.Beckhoff_EKx9xx.Beckhoff_EKx9xxEK1122.A_0008_EK1960_2608_0021.Module_1_FSoE.FSoE_Outputs.FSOE/FSIN_Module_10_Err_Ack_2 <-> Module 1 (FSoE)/FSoE Outputs/FSOE/FSIN Module 10.Err Ack 2
//     PlcTask Outputs/GVL_iXlinker.EtherCAT_Master_EKxxxx.Beckhoff_EKx9xx.Beckhoff_EKx9xxEK1122.A_0008_EK1960_2608_0021.Module_1_FSoE.FSoE_Outputs.FSOE/FSoE_Connection_ID <-> Module 1 (FSoE)/FSoE Outputs/FSOE/FSoE Connection ID
//     PlcTask Outputs/GVL_iXlinker.EtherCAT_Master_EKxxxx.Beckhoff_EKx9xx.Beckhoff_EKx9xxEK1122.A_0008_EK1960_2608_0021.Module_2_FSOUT.Outputs.Module_1_Channel_1_Standard_Output_X5_1 <-> Module 2 (FSOUT)/Outputs/Module 1.Channel 1.Standard Output (X5.1)
//     PlcTask Outputs/GVL_iXlinker.EtherCAT_Master_EKxxxx.Beckhoff_EKx9xx.Beckhoff_EKx9xxEK1122.A_0008_EK1960_2608_0021.Module_2_FSOUT.Outputs.Module_1_Channel_2_Standard_Output_X5_2 <-> Module 2 (FSOUT)/Outputs/Module 1.Channel 2.Standard Output (X5.2)
//     PlcTask Outputs/GVL_iXlinker.EtherCAT_Master_EKxxxx.Beckhoff_EKx9xx.Beckhoff_EKx9xxEK1122.A_0008_EK1960_2608_0021.Module_2_FSOUT.Outputs.Module_1_Channel_3_Standard_Output_X5_3 <-> Module 2 (FSOUT)/Outputs/Module 1.Channel 3.Standard Output (X5.3)
//     PlcTask Outputs/GVL_iXlinker.EtherCAT_Master_EKxxxx.Beckhoff_EKx9xx.Beckhoff_EKx9xxEK1122.A_0008_EK1960_2608_0021.Module_2_FSOUT.Outputs.Module_1_Channel_4_Standard_Output_X5_4 <-> Module 2 (FSOUT)/Outputs/Module 1.Channel 4.Standard Output (X5.4)
//     PlcTask Outputs/GVL_iXlinker.EtherCAT_Master_EKxxxx.Beckhoff_EKx9xx.Beckhoff_EKx9xxEK1122.A_0008_EK1960_2608_0021.Module_2_FSOUT.Outputs.Module_2_Channel_1_Standard_Output_X5_5 <-> Module 2 (FSOUT)/Outputs/Module 2.Channel 1.Standard Output (X5.5)
//     PlcTask Outputs/GVL_iXlinker.EtherCAT_Master_EKxxxx.Beckhoff_EKx9xx.Beckhoff_EKx9xxEK1122.A_0008_EK1960_2608_0021.Module_2_FSOUT.Outputs.Module_2_Channel_2_Standard_Output_X5_6 <-> Module 2 (FSOUT)/Outputs/Module 2.Channel 2.Standard Output (X5.6)
//     PlcTask Outputs/GVL_iXlinker.EtherCAT_Master_EKxxxx.Beckhoff_EKx9xx.Beckhoff_EKx9xxEK1122.A_0008_EK1960_2608_0021.Module_2_FSOUT.Outputs.Module_2_Channel_3_Standard_Output_X5_7 <-> Module 2 (FSOUT)/Outputs/Module 2.Channel 3.Standard Output (X5.7)
//     PlcTask Outputs/GVL_iXlinker.EtherCAT_Master_EKxxxx.Beckhoff_EKx9xx.Beckhoff_EKx9xxEK1122.A_0008_EK1960_2608_0021.Module_2_FSOUT.Outputs.Module_2_Channel_4_Standard_Output_X5_8 <-> Module 2 (FSOUT)/Outputs/Module 2.Channel 4.Standard Output (X5.8)
//     PlcTask Outputs/GVL_iXlinker.EtherCAT_Master_EKxxxx.Beckhoff_EKx9xx.Beckhoff_EKx9xxEK1122.A_0008_EK1960_2608_0021.Module_2_FSOUT.Outputs.Module_3_Channel_1_Standard_Output_X7_1 <-> Module 2 (FSOUT)/Outputs/Module 3.Channel 1.Standard Output (X7.1)
//     PlcTask Outputs/GVL_iXlinker.EtherCAT_Master_EKxxxx.Beckhoff_EKx9xx.Beckhoff_EKx9xxEK1122.A_0008_EK1960_2608_0021.Module_2_FSOUT.Outputs.Module_3_Channel_2_Standard_Output_X7_2 <-> Module 2 (FSOUT)/Outputs/Module 3.Channel 2.Standard Output (X7.2)
//     PlcTask Outputs/GVL_iXlinker.EtherCAT_Master_EKxxxx.Beckhoff_EKx9xx.Beckhoff_EKx9xxEK1122.A_0008_EK1960_2608_0021.Module_2_FSOUT.Outputs.Module_3_Channel_3_Standard_Output_X7_3 <-> Module 2 (FSOUT)/Outputs/Module 3.Channel 3.Standard Output (X7.3)
//     PlcTask Outputs/GVL_iXlinker.EtherCAT_Master_EKxxxx.Beckhoff_EKx9xx.Beckhoff_EKx9xxEK1122.A_0008_EK1960_2608_0021.Module_2_FSOUT.Outputs.Module_3_Channel_4_Standard_Output_X7_4 <-> Module 2 (FSOUT)/Outputs/Module 3.Channel 4.Standard Output (X7.4)
//     PlcTask Outputs/GVL_iXlinker.EtherCAT_Master_EKxxxx.Beckhoff_EKx9xx.Beckhoff_EKx9xxEK1122.A_0008_EK1960_2608_0021.Module_2_FSOUT.Outputs.Module_4_Channel_1_Standard_Output_X7_5 <-> Module 2 (FSOUT)/Outputs/Module 4.Channel 1.Standard Output (X7.5)
//     PlcTask Outputs/GVL_iXlinker.EtherCAT_Master_EKxxxx.Beckhoff_EKx9xx.Beckhoff_EKx9xxEK1122.A_0008_EK1960_2608_0021.Module_2_FSOUT.Outputs.Module_4_Channel_2_Standard_Output_X7_6 <-> Module 2 (FSOUT)/Outputs/Module 4.Channel 2.Standard Output (X7.6)
//     PlcTask Outputs/GVL_iXlinker.EtherCAT_Master_EKxxxx.Beckhoff_EKx9xx.Beckhoff_EKx9xxEK1122.A_0008_EK1960_2608_0021.Module_2_FSOUT.Outputs.Module_4_Channel_3_Standard_Output_X7_7 <-> Module 2 (FSOUT)/Outputs/Module 4.Channel 3.Standard Output (X7.7)
//     PlcTask Outputs/GVL_iXlinker.EtherCAT_Master_EKxxxx.Beckhoff_EKx9xx.Beckhoff_EKx9xxEK1122.A_0008_EK1960_2608_0021.Module_2_FSOUT.Outputs.Module_4_Channel_4_Standard_Output_X7_8 <-> Module 2 (FSOUT)/Outputs/Module 4.Channel 4.Standard Output (X7.8)
//     PlcTask Outputs/GVL_iXlinker.EtherCAT_Master_EKxxxx.Beckhoff_EKx9xx.Beckhoff_EKx9xxEK1122.A_0008_EK1960_2608_0021.Module_2_FSOUT.Outputs.Module_5_Channel_1_Standard_Output_X9_1 <-> Module 2 (FSOUT)/Outputs/Module 5.Channel 1.Standard Output (X9.1)
//     PlcTask Outputs/GVL_iXlinker.EtherCAT_Master_EKxxxx.Beckhoff_EKx9xx.Beckhoff_EKx9xxEK1122.A_0008_EK1960_2608_0021.Module_2_FSOUT.Outputs.Module_5_Channel_2_Standard_Output_X9_2 <-> Module 2 (FSOUT)/Outputs/Module 5.Channel 2.Standard Output (X9.2)
//     PlcTask Outputs/GVL_iXlinker.EtherCAT_Master_EKxxxx.Beckhoff_EKx9xx.Beckhoff_EKx9xxEK1122.A_0008_EK1960_2608_0021.Module_2_FSOUT.Outputs.Module_5_Channel_3_Standard_Output_X9_3 <-> Module 2 (FSOUT)/Outputs/Module 5.Channel 3.Standard Output (X9.3)
//     PlcTask Outputs/GVL_iXlinker.EtherCAT_Master_EKxxxx.Beckhoff_EKx9xx.Beckhoff_EKx9xxEK1122.A_0008_EK1960_2608_0021.Module_2_FSOUT.Outputs.Module_5_Channel_4_Standard_Output_X9_4 <-> Module 2 (FSOUT)/Outputs/Module 5.Channel 4.Standard Output (X9.4)
//     PlcTask Outputs/GVL_iXlinker.EtherCAT_Master_EKxxxx.Beckhoff_EKx9xx.Beckhoff_EKx9xxEK1122.A_0008_EK1960_2608_0021.Module_2_FSOUT.Outputs.Module_6_Channel_1_Standard_Output_X9_5 <-> Module 2 (FSOUT)/Outputs/Module 6.Channel 1.Standard Output (X9.5)
//     PlcTask Outputs/GVL_iXlinker.EtherCAT_Master_EKxxxx.Beckhoff_EKx9xx.Beckhoff_EKx9xxEK1122.A_0008_EK1960_2608_0021.Module_2_FSOUT.Outputs.Module_6_Channel_2_Standard_Output_X9_6 <-> Module 2 (FSOUT)/Outputs/Module 6.Channel 2.Standard Output (X9.6)
//     PlcTask Outputs/GVL_iXlinker.EtherCAT_Master_EKxxxx.Beckhoff_EKx9xx.Beckhoff_EKx9xxEK1122.A_0008_EK1960_2608_0021.Module_2_FSOUT.Outputs.Module_6_Channel_3_Standard_Output_X9_7 <-> Module 2 (FSOUT)/Outputs/Module 6.Channel 3.Standard Output (X9.7)
//     PlcTask Outputs/GVL_iXlinker.EtherCAT_Master_EKxxxx.Beckhoff_EKx9xx.Beckhoff_EKx9xxEK1122.A_0008_EK1960_2608_0021.Module_2_FSOUT.Outputs.Module_6_Channel_4_Standard_Output_X9_8 <-> Module 2 (FSOUT)/Outputs/Module 6.Channel 4.Standard Output (X9.8)
//     PlcTask Outputs/GVL_iXlinker.EtherCAT_Master_EKxxxx.Beckhoff_EKx9xx.Beckhoff_EKx9xxEK1122.A_0008_EK1960_2608_0021.Module_2_FSOUT.Outputs.Relais_Module_Channel_1_Standard_Output_X4_1_X4_5 <-> Module 2 (FSOUT)/Outputs/Relais Module.Channel 1.Standard Output (X4.1, X4.5)
//     PlcTask Outputs/GVL_iXlinker.EtherCAT_Master_EKxxxx.Beckhoff_EKx9xx.Beckhoff_EKx9xxEK1122.A_0008_EK1960_2608_0021.Module_2_FSOUT.Outputs.Relais_Module_Channel_2_Standard_Output_X4_2_X4_6 <-> Module 2 (FSOUT)/Outputs/Relais Module.Channel 2.Standard Output (X4.2, X4.6)
//     PlcTask Outputs/GVL_iXlinker.EtherCAT_Master_EKxxxx.Beckhoff_EKx9xx.Beckhoff_EKx9xxEK1122.A_0008_EK1960_2608_0021.Module_2_FSOUT.Outputs.Relais_Module_Channel_3_Standard_Output_X4_3_X4_7 <-> Module 2 (FSOUT)/Outputs/Relais Module.Channel 3.Standard Output (X4.3, X4.7)
//     PlcTask Outputs/GVL_iXlinker.EtherCAT_Master_EKxxxx.Beckhoff_EKx9xx.Beckhoff_EKx9xxEK1122.A_0008_EK1960_2608_0021.Module_2_FSOUT.Outputs.Relais_Module_Channel_4_Standard_Output_X4_4_X4_8 <-> Module 2 (FSOUT)/Outputs/Relais Module.Channel 4.Standard Output (X4.4, X4.8)
//     PlcTask Inputs/GVL_iXlinker.EtherCAT_Master_EKxxxx.Beckhoff_EKx9xx.Beckhoff_EKx9xxEK1122.A_0008_EK1960_2608_0021.Module_3_FSLOGIC.FSLOGIC_Inputs.Safe_Logic_State <-> Module 3 (FSLOGIC)/FSLOGIC Inputs/Safe Logic State
//     PlcTask Inputs/GVL_iXlinker.EtherCAT_Master_EKxxxx.Beckhoff_EKx9xx.Beckhoff_EKx9xxEK1122.A_0008_EK1960_2608_0021.Module_3_FSLOGIC.FSLOGIC_Inputs.Cycle_Counter <-> Module 3 (FSLOGIC)/FSLOGIC Inputs/Cycle Counter
//     PlcTask Inputs/GVL_iXlinker.EtherCAT_Master_EKxxxx.Beckhoff_EKx9xx.Beckhoff_EKx9xxEK1122.A_0008_EK1960_2608_0021.WcState.WcState0 <-> WcState/WcState0
//     PlcTask Inputs/GVL_iXlinker.EtherCAT_Master_EKxxxx.Beckhoff_EKx9xx.Beckhoff_EKx9xxEK1122.A_0008_EK1960_2608_0021.WcState.WcState1 <-> WcState/WcState1
//     PlcTask Inputs/GVL_iXlinker.EtherCAT_Master_EKxxxx.Beckhoff_EKx9xx.Beckhoff_EKx9xxEK1122.A_0008_EK1960_2608_0021.WcState.InputToggle0 <-> WcState/InputToggle0
//     PlcTask Inputs/GVL_iXlinker.EtherCAT_Master_EKxxxx.Beckhoff_EKx9xx.Beckhoff_EKx9xxEK1122.A_0008_EK1960_2608_0021.WcState.InputToggle1 <-> WcState/InputToggle1
//     PlcTask Inputs/GVL_iXlinker.EtherCAT_Master_EKxxxx.Beckhoff_EKx9xx.Beckhoff_EKx9xxEK1122.A_0008_EK1960_2608_0021.InfoData.AdsAddr <-> InfoData/AdsAddr
//     PlcTask Inputs/GVL_iXlinker.EtherCAT_Master_EKxxxx.Beckhoff_EKx9xx.Beckhoff_EKx9xxEK1122.A_0008_EK1960_2608_0021.InfoData.State <-> InfoData/State
//   PLC/PLC Instance <-> EtherCAT Master EKxxxx/Beckhoff EKxxxx-0080
//     PlcTask Inputs/GVL_iXlinker.EtherCAT_Master_EKxxxx.Beckhoff_EKxxxx_0080.InfoData.State <-> InfoData/State
//   PLC/PLC Instance <-> EtherCAT Master EKxxxx/Beckhoff EKxxxx-0080/Beckhoff EKxxxx-0080EK1122
//     PlcTask Inputs/GVL_iXlinker.EtherCAT_Master_EKxxxx.Beckhoff_EKxxxx_0080.Beckhoff_EKxxxx_0080EK1122.InfoData.State <-> InfoData/State
//   PLC/PLC Instance <-> EtherCAT Master EKxxxx/Beckhoff EKxxxx-0080/Beckhoff EKxxxx-0080EK1122/Beckhoff EKxxxx-0080sub EK1100
//     PlcTask Inputs/GVL_iXlinker.EtherCAT_Master_EKxxxx.Beckhoff_EKxxxx_0080.Beckhoff_EKxxxx_0080EK1122.Beckhoff_EKxxxx_0080sub_EK1100.InfoData.State <-> InfoData/State
//   PLC/PLC Instance <-> EtherCAT Master EKxxxx/Beckhoff EKxxxx-0080/A_0006(EK1122-0080-0019)
//     PlcTask Inputs/GVL_iXlinker.EtherCAT_Master_EKxxxx.Beckhoff_EKxxxx_0080.A_0006_EK1122_0080_0019.InfoData.State <-> InfoData/State
//   PLC/PLC Instance <-> EtherCAT Master EKxxxx/Beckhoff EKxxxx-0080/A_0005(EK1122-0080-0018)
//     PlcTask Inputs/GVL_iXlinker.EtherCAT_Master_EKxxxx.Beckhoff_EKxxxx_0080.A_0005_EK1122_0080_0018.InfoData.State <-> InfoData/State
//   PLC/PLC Instance <-> EtherCAT Master EKxxxx/Beckhoff EKxxxx-0080/A_0004(EK1122-0080-0017)
//     PlcTask Inputs/GVL_iXlinker.EtherCAT_Master_EKxxxx.Beckhoff_EKxxxx_0080.A_0004_EK1122_0080_0017.InfoData.State <-> InfoData/State
//   PLC/PLC Instance <-> EtherCAT_Master_EKxxxx
//     PlcTask Inputs/GVL_iXlinker.EtherCAT_Master_EKxxxx.SyncUnits._default._unreferenced.WcState.WcState <-> SyncUnits/<default>/<unreferenced>/WcState/WcState
//     PlcTask Inputs/GVL_iXlinker.EtherCAT_Master_EKxxxx.SyncUnits._default._unreferenced.InfoData.ObjectId <-> SyncUnits/<default>/<unreferenced>/InfoData/ObjectId
//     PlcTask Inputs/GVL_iXlinker.EtherCAT_Master_EKxxxx.SyncUnits._default._unreferenced.InfoData.State <-> SyncUnits/<default>/<unreferenced>/InfoData/State
//     PlcTask Inputs/GVL_iXlinker.EtherCAT_Master_EKxxxx.SyncUnits._default._unreferenced.InfoData.SlaveCount <-> SyncUnits/<default>/<unreferenced>/InfoData/SlaveCount
//     PlcTask Inputs/GVL_iXlinker.EtherCAT_Master_EKxxxx.SyncUnits._default.PlcTask.WcState.WcState <-> SyncUnits/<default>/PlcTask/WcState/WcState
//     PlcTask Inputs/GVL_iXlinker.EtherCAT_Master_EKxxxx.SyncUnits._default.PlcTask.InfoData.ObjectId <-> SyncUnits/<default>/PlcTask/InfoData/ObjectId
//     PlcTask Inputs/GVL_iXlinker.EtherCAT_Master_EKxxxx.SyncUnits._default.PlcTask.InfoData.State <-> SyncUnits/<default>/PlcTask/InfoData/State
//     PlcTask Inputs/GVL_iXlinker.EtherCAT_Master_EKxxxx.SyncUnits._default.PlcTask.InfoData.SlaveCount <-> SyncUnits/<default>/PlcTask/InfoData/SlaveCount
//     PlcTask Inputs/GVL_iXlinker.EtherCAT_Master_EKxxxx.Inputs.SlaveCount <-> Inputs/SlaveCount
//     PlcTask Inputs/GVL_iXlinker.EtherCAT_Master_EKxxxx.Inputs.DevState <-> Inputs/DevState
//     PlcTask Inputs/GVL_iXlinker.EtherCAT_Master_EKxxxx.Inputs.Frm{0..25}State <-> Inputs/Frm{0..25}State  (26 links)
//     PlcTask Inputs/GVL_iXlinker.EtherCAT_Master_EKxxxx.Inputs.Frm{0..25}WcState <-> Inputs/Frm{0..25}WcState  (26 links)
//     PlcTask Inputs/GVL_iXlinker.EtherCAT_Master_EKxxxx.Inputs.Frm{0..25}InputToggle <-> Inputs/Frm{0..25}InputToggle  (26 links)
//     PlcTask Outputs/GVL_iXlinker.EtherCAT_Master_EKxxxx.Outputs.DevCtrl <-> Outputs/DevCtrl
//     PlcTask Outputs/GVL_iXlinker.EtherCAT_Master_EKxxxx.Outputs.Frm{0..25}Ctrl <-> Outputs/Frm{0..25}Ctrl  (26 links)
//     PlcTask Outputs/GVL_iXlinker.EtherCAT_Master_EKxxxx.Outputs.Frm{0..25}WcCtrl <-> Outputs/Frm{0..25}WcCtrl  (26 links)
//     PlcTask Inputs/GVL_iXlinker.EtherCAT_Master_EKxxxx.InfoData.ChangeCount <-> InfoData/ChangeCount
//     PlcTask Inputs/GVL_iXlinker.EtherCAT_Master_EKxxxx.InfoData.DevId <-> InfoData/DevId
//     PlcTask Inputs/GVL_iXlinker.EtherCAT_Master_EKxxxx.InfoData.AmsNetId <-> InfoData/AmsNetId
//     PlcTask Inputs/GVL_iXlinker.EtherCAT_Master_EKxxxx.InfoData.CfgSlaveCount <-> InfoData/CfgSlaveCount
//     PlcTask Inputs/GVL_iXlinker.EtherCAT_Master_EKxxxx.InfoData.DcToTcTimeOffset <-> InfoData/DcToTcTimeOffset
//     PlcTask Inputs/GVL_iXlinker.EtherCAT_Master_EKxxxx.InfoData.DcToExtTimeOffset <-> InfoData/DcToExtTimeOffset

CONFIGURATION PLC
    RESOURCE PLC ON TwinCAT3
        TASK PlcTask(INTERVAL := T#10ms, PRIORITY := 20);
        PROGRAM MAIN WITH PlcTask : MAIN;
    END_RESOURCE
END_CONFIGURATION

// ---- DUTs/IO/PdoEntries/Status_9847B4EF.TcDUT
{attribute 'GeneratedUsingTerminal: EKM1101-0000-0016'}
{attribute addProperty BoxType "EKM1101-0000-0016"}
{attribute addProperty Id "DiagBOOL1ErrorBOOL1Input_cycle_CounterBYTE1TxPDO_StateBOOL1IDUSINT1"}
{attribute addProperty CRC "2554836207"}
{attribute addProperty Size "5"}
TYPE Status_9847B4EF :
STRUCT
	{attribute addProperty Name "Diag"}
	Diag : BOOL;
	{attribute addProperty Name "Error"}
	Error : BOOL;
	{attribute addProperty Name "Input_cycle_Counter"}
	Input_cycle_Counter : BYTE;
	{attribute addProperty Name "TxPDO_State"}
	TxPDO_State : BOOL;
	{attribute addProperty Name "ID"}
	ID : USINT;
END_STRUCT
END_TYPE

// ---- DUTs/IO/PdoEntries/Status_BA3D1C5D.TcDUT
{attribute 'GeneratedUsingTerminal: EKM1101-0000-0016'}
{attribute addProperty BoxType "EKM1101-0000-0016"}
{attribute addProperty Id "ErrorBOOL1UnderrangeBOOL1OverrangeBOOL1DiagBOOL1Sensor_OvrBOOL1OverrunBOOL1TxPDO_StateBOOL1"}
{attribute addProperty CRC "3124567133"}
{attribute addProperty Size "7"}
TYPE Status_BA3D1C5D :
STRUCT
	{attribute addProperty Name "Error"}
	Error : BOOL;
	{attribute addProperty Name "Underrange"}
	Underrange : BOOL;
	{attribute addProperty Name "Overrange"}
	Overrange : BOOL;
	{attribute addProperty Name "Diag"}
	Diag : BOOL;
	{attribute addProperty Name "Sensor_Ovr"}
	Sensor_Ovr : BOOL;
	{attribute addProperty Name "Overrun"}
	Overrun : BOOL;
	{attribute addProperty Name "TxPDO_State"}
	TxPDO_State : BOOL;
END_STRUCT
END_TYPE

// ---- DUTs/IO/PdoEntries/Status_F2CE6D91.TcDUT
{attribute 'GeneratedUsingTerminal: EKM1101-0000-0016'}
{attribute addProperty BoxType "EKM1101-0000-0016"}
{attribute addProperty Id "UnderrangeBOOL1OverrangeBOOL1Limit_1BYTE1Limit_2BYTE1ErrorBOOL1TxPDO_StateBOOL1TxPDO_ToggleBOOL1"}
{attribute addProperty CRC "4073614737"}
{attribute addProperty Size "7"}
TYPE Status_F2CE6D91 :
STRUCT
	{attribute addProperty Name "Underrange"}
	Underrange : BOOL;
	{attribute addProperty Name "Overrange"}
	Overrange : BOOL;
	{attribute addProperty Name "Limit_1"}
	Limit_1 : BYTE;
	{attribute addProperty Name "Limit_2"}
	Limit_2 : BYTE;
	{attribute addProperty Name "Error"}
	Error : BOOL;
	{attribute addProperty Name "TxPDO_State"}
	TxPDO_State : BOOL;
	{attribute addProperty Name "TxPDO_Toggle"}
	TxPDO_Toggle : BOOL;
END_STRUCT
END_TYPE

// ---- DUTs/IO/PdoEntries/Control_EBEDCF76.TcDUT
{attribute 'GeneratedUsingTerminal: EKM1101-0000-0016'}
{attribute addProperty BoxType "EKM1101-0000-0016"}
{attribute addProperty Id "Up_Out_OFFBOOL1"}
{attribute addProperty CRC "3958230902"}
{attribute addProperty Size "1"}
TYPE Control_EBEDCF76 :
STRUCT
	{attribute addProperty Name "Up_Out_OFF"}
	Up_Out_OFF : BOOL;
END_STRUCT
END_TYPE

// ---- DUTs/IO/PdoEntries/FSOE_BBDEEE9E.TcDUT
{attribute 'GeneratedUsingTerminal: EK1960-0000-0019'}
{attribute addProperty BoxType "EK1960-0000-0019"}
{attribute addProperty Id "FSoE_CommandUSINT1FSOUT_Module_1_Module_FaultBOOL1FSOUT_Module_2_Module_FaultBOOL1FSOUT_Module_3_Module_FaultBOOL1FSOUT_Module_4_Module_FaultBOOL1FSOUT_Module_5_Module_FaultBOOL1FSOUT_Module_6_Module_FaultBOOL1FSIN_Module_1_Channel_1_InputBOOL1FSIN_Module_1_Channel_2_InputBOOL1FSIN_Module_1_Module_FaultBOOL1FSIN_Module_2_Channel_1_InputBOOL1FSIN_Module_2_Channel_2_InputBOOL1FSIN_Module_2_Module_FaultBOOL1FSIN_Module_3_Channel_1_InputBOOL1FSIN_Module_3_Channel_2_InputBOOL1FSIN_Module_3_Module_FaultBOOL1FSoE_CRC_000UINT2FSIN_Module_4_Channel_1_InputBOOL1FSIN_Module_4_Channel_2_InputBOOL1FSIN_Module_4_Module_FaultBOOL1FSIN_Module_5_Channel_1_InputBOOL1FSIN_Module_5_Channel_2_InputBOOL1FSIN_Module_5_Module_FaultBOOL1FSIN_Module_6_Channel_1_InputBOOL1FSIN_Module_6_Channel_2_InputBOOL1FSIN_Module_6_Module_FaultBOOL1FSIN_Module_7_Channel_1_InputBOOL1FSIN_Module_7_Channel_2_InputBOOL1FSIN_Module_7_Module_FaultBOOL1FSIN_Module_8_Channel_1_InputBOOL1FSIN_Module_8_Channel_2_InputBOOL1FSIN_Module_8_Module_FaultBOOL1FSIN_Module_9_Channel_1_InputBOOL1FSoE_CRC_001UINT2FSIN_Module_9_Channel_2_InputBOOL1FSIN_Module_9_Module_Fault_1BOOL1FSIN_Module_9_Module_Fault_2BOOL1FSIN_Module_10_Channel_1_InputBOOL1FSIN_Module_10_Channel_2_InputBOOL1FSIN_Module_10_Module_Fault_1BOOL1FSIN_Module_10_Module_Fault_2BOOL1FSoE_CRC_002UINT2FSoE_Connection_IDUINT2"}
{attribute addProperty CRC "3151949470"}
{attribute addProperty Size "47"}
TYPE FSOE_BBDEEE9E :
STRUCT
	{attribute addProperty Name "FSoE_Command"}
	FSoE_Command : USINT;
	{attribute addProperty Name "FSOUT_Module_1_Module_Fault"}
	FSOUT_Module_1_Module_Fault : BOOL;
	{attribute addProperty Name "FSOUT_Module_2_Module_Fault"}
	FSOUT_Module_2_Module_Fault : BOOL;
	{attribute addProperty Name "FSOUT_Module_3_Module_Fault"}
	FSOUT_Module_3_Module_Fault : BOOL;
	{attribute addProperty Name "FSOUT_Module_4_Module_Fault"}
	FSOUT_Module_4_Module_Fault : BOOL;
	{attribute addProperty Name "FSOUT_Module_5_Module_Fault"}
	FSOUT_Module_5_Module_Fault : BOOL;
	{attribute addProperty Name "FSOUT_Module_6_Module_Fault"}
	FSOUT_Module_6_Module_Fault : BOOL;
	{attribute addProperty Name "FSIN_Module_1_Channel_1_Input"}
	FSIN_Module_1_Channel_1_Input : BOOL;
	{attribute addProperty Name "FSIN_Module_1_Channel_2_Input"}
	FSIN_Module_1_Channel_2_Input : BOOL;
	{attribute addProperty Name "FSIN_Module_1_Module_Fault"}
	FSIN_Module_1_Module_Fault : BOOL;
	{attribute addProperty Name "FSIN_Module_2_Channel_1_Input"}
	FSIN_Module_2_Channel_1_Input : BOOL;
	{attribute addProperty Name "FSIN_Module_2_Channel_2_Input"}
	FSIN_Module_2_Channel_2_Input : BOOL;
	{attribute addProperty Name "FSIN_Module_2_Module_Fault"}
	FSIN_Module_2_Module_Fault : BOOL;
	{attribute addProperty Name "FSIN_Module_3_Channel_1_Input"}
	FSIN_Module_3_Channel_1_Input : BOOL;
	{attribute addProperty Name "FSIN_Module_3_Channel_2_Input"}
	FSIN_Module_3_Channel_2_Input : BOOL;
	{attribute addProperty Name "FSIN_Module_3_Module_Fault"}
	FSIN_Module_3_Module_Fault : BOOL;
	{attribute addProperty Name "FSoE_CRC_000"}
	FSoE_CRC_000 : UINT;
	{attribute addProperty Name "FSIN_Module_4_Channel_1_Input"}
	FSIN_Module_4_Channel_1_Input : BOOL;
	{attribute addProperty Name "FSIN_Module_4_Channel_2_Input"}
	FSIN_Module_4_Channel_2_Input : BOOL;
	{attribute addProperty Name "FSIN_Module_4_Module_Fault"}
	FSIN_Module_4_Module_Fault : BOOL;
	{attribute addProperty Name "FSIN_Module_5_Channel_1_Input"}
	FSIN_Module_5_Channel_1_Input : BOOL;
	{attribute addProperty Name "FSIN_Module_5_Channel_2_Input"}
	FSIN_Module_5_Channel_2_Input : BOOL;
	{attribute addProperty Name "FSIN_Module_5_Module_Fault"}
	FSIN_Module_5_Module_Fault : BOOL;
	{attribute addProperty Name "FSIN_Module_6_Channel_1_Input"}
	FSIN_Module_6_Channel_1_Input : BOOL;
	{attribute addProperty Name "FSIN_Module_6_Channel_2_Input"}
	FSIN_Module_6_Channel_2_Input : BOOL;
	{attribute addProperty Name "FSIN_Module_6_Module_Fault"}
	FSIN_Module_6_Module_Fault : BOOL;
	{attribute addProperty Name "FSIN_Module_7_Channel_1_Input"}
	FSIN_Module_7_Channel_1_Input : BOOL;
	{attribute addProperty Name "FSIN_Module_7_Channel_2_Input"}
	FSIN_Module_7_Channel_2_Input : BOOL;
	{attribute addProperty Name "FSIN_Module_7_Module_Fault"}
	FSIN_Module_7_Module_Fault : BOOL;
	{attribute addProperty Name "FSIN_Module_8_Channel_1_Input"}
	FSIN_Module_8_Channel_1_Input : BOOL;
	{attribute addProperty Name "FSIN_Module_8_Channel_2_Input"}
	FSIN_Module_8_Channel_2_Input : BOOL;
	{attribute addProperty Name "FSIN_Module_8_Module_Fault"}
	FSIN_Module_8_Module_Fault : BOOL;
	{attribute addProperty Name "FSIN_Module_9_Channel_1_Input"}
	FSIN_Module_9_Channel_1_Input : BOOL;
	{attribute addProperty Name "FSoE_CRC_001"}
	FSoE_CRC_001 : UINT;
	{attribute addProperty Name "FSIN_Module_9_Channel_2_Input"}
	FSIN_Module_9_Channel_2_Input : BOOL;
	{attribute addProperty Name "FSIN_Module_9_Module_Fault_1"}
	FSIN_Module_9_Module_Fault_1 : BOOL;
	{attribute addProperty Name "FSIN_Module_9_Module_Fault_2"}
	FSIN_Module_9_Module_Fault_2 : BOOL;
	{attribute addProperty Name "FSIN_Module_10_Channel_1_Input"}
	FSIN_Module_10_Channel_1_Input : BOOL;
	{attribute addProperty Name "FSIN_Module_10_Channel_2_Input"}
	FSIN_Module_10_Channel_2_Input : BOOL;
	{attribute addProperty Name "FSIN_Module_10_Module_Fault_1"}
	FSIN_Module_10_Module_Fault_1 : BOOL;
	{attribute addProperty Name "FSIN_Module_10_Module_Fault_2"}
	FSIN_Module_10_Module_Fault_2 : BOOL;
	{attribute addProperty Name "FSoE_CRC_002"}
	FSoE_CRC_002 : UINT;
	{attribute addProperty Name "FSoE_Connection_ID"}
	FSoE_Connection_ID : UINT;
END_STRUCT
END_TYPE

// ---- DUTs/IO/PdoEntries/FSOE_BAC7BF21.TcDUT
{attribute 'GeneratedUsingTerminal: EK1960-0000-0019'}
{attribute addProperty BoxType "EK1960-0000-0019"}
{attribute addProperty Id "FSoE_CommandUSINT1FSOUT_Module_1_Channel_1_OutputBOOL1FSOUT_Module_1_Channel_2_OutputBOOL1FSOUT_Module_1_Channel_3_OutputBOOL1FSOUT_Module_1_Channel_4_OutputBOOL1FSOUT_Module_1_ErrAckBOOL1FSOUT_Module_2_Channel_1_OutputBOOL1FSOUT_Module_2_Channel_2_OutputBOOL1FSOUT_Module_2_Channel_3_OutputBOOL1FSOUT_Module_2_Channel_4_OutputBOOL1FSOUT_Module_2_ErrAckBOOL1FSOUT_Module_3_Channel_1_OutputBOOL1FSOUT_Module_3_Channel_2_OutputBOOL1FSOUT_Module_3_Channel_3_OutputBOOL1FSOUT_Module_3_Channel_4_OutputBOOL1FSOUT_Module_3_ErrAckBOOL1FSOUT_Module_4_Channel_1_OutputBOOL1FSoE_CRC_000UINT2FSOUT_Module_4_Channel_2_OutputBOOL1FSOUT_Module_4_Channel_3_OutputBOOL1FSOUT_Module_4_Channel_4_OutputBOOL1FSOUT_Module_4_ErrAckBOOL1FSOUT_Module_5_Channel_1_OutputBOOL1FSOUT_Module_5_Channel_2_OutputBOOL1FSOUT_Module_5_Channel_3_OutputBOOL1FSOUT_Module_5_Channel_4_OutputBOOL1FSOUT_Module_5_ErrAckBOOL1FSOUT_Module_6_Channel_1_OutputBOOL1FSOUT_Module_6_Channel_2_OutputBOOL1FSOUT_Module_6_Channel_3_OutputBOOL1FSOUT_Module_6_Channel_4_OutputBOOL1FSOUT_Module_6_ErrAckBOOL1FSoE_CRC_001UINT2FSIN_Module_1_ErrAckBOOL1FSIN_Module_2_ErrAckBOOL1FSIN_Module_3_ErrAckBOOL1FSIN_Module_4_ErrAckBOOL1FSIN_Module_5_ErrAckBOOL1FSIN_Module_6_ErrAckBOOL1FSIN_Module_7_ErrAckBOOL1FSIN_Module_8_ErrAckBOOL1FSIN_Module_9_ErrAck_1BOOL1FSIN_Module_9_ErrAck_2BOOL1FSIN_Module_10_ErrAck_1BOOL1FSIN_Module_10_ErrAck_2BOOL1FSoE_CRC_002UINT2FSoE_Connection_IDUINT2"}
{attribute addProperty CRC "3133652769"}
{attribute addProperty Size "51"}
TYPE FSOE_BAC7BF21 :
STRUCT
	{attribute addProperty Name "FSoE_Command"}
	FSoE_Command : USINT;
	{attribute addProperty Name "FSOUT_Module_1_Channel_1_Output"}
	FSOUT_Module_1_Channel_1_Output : BOOL;
	{attribute addProperty Name "FSOUT_Module_1_Channel_2_Output"}
	FSOUT_Module_1_Channel_2_Output : BOOL;
	{attribute addProperty Name "FSOUT_Module_1_Channel_3_Output"}
	FSOUT_Module_1_Channel_3_Output : BOOL;
	{attribute addProperty Name "FSOUT_Module_1_Channel_4_Output"}
	FSOUT_Module_1_Channel_4_Output : BOOL;
	{attribute addProperty Name "FSOUT_Module_1_ErrAck"}
	FSOUT_Module_1_ErrAck : BOOL;
	{attribute addProperty Name "FSOUT_Module_2_Channel_1_Output"}
	FSOUT_Module_2_Channel_1_Output : BOOL;
	{attribute addProperty Name "FSOUT_Module_2_Channel_2_Output"}
	FSOUT_Module_2_Channel_2_Output : BOOL;
	{attribute addProperty Name "FSOUT_Module_2_Channel_3_Output"}
	FSOUT_Module_2_Channel_3_Output : BOOL;
	{attribute addProperty Name "FSOUT_Module_2_Channel_4_Output"}
	FSOUT_Module_2_Channel_4_Output : BOOL;
	{attribute addProperty Name "FSOUT_Module_2_ErrAck"}
	FSOUT_Module_2_ErrAck : BOOL;
	{attribute addProperty Name "FSOUT_Module_3_Channel_1_Output"}
	FSOUT_Module_3_Channel_1_Output : BOOL;
	{attribute addProperty Name "FSOUT_Module_3_Channel_2_Output"}
	FSOUT_Module_3_Channel_2_Output : BOOL;
	{attribute addProperty Name "FSOUT_Module_3_Channel_3_Output"}
	FSOUT_Module_3_Channel_3_Output : BOOL;
	{attribute addProperty Name "FSOUT_Module_3_Channel_4_Output"}
	FSOUT_Module_3_Channel_4_Output : BOOL;
	{attribute addProperty Name "FSOUT_Module_3_ErrAck"}
	FSOUT_Module_3_ErrAck : BOOL;
	{attribute addProperty Name "FSOUT_Module_4_Channel_1_Output"}
	FSOUT_Module_4_Channel_1_Output : BOOL;
	{attribute addProperty Name "FSoE_CRC_000"}
	FSoE_CRC_000 : UINT;
	{attribute addProperty Name "FSOUT_Module_4_Channel_2_Output"}
	FSOUT_Module_4_Channel_2_Output : BOOL;
	{attribute addProperty Name "FSOUT_Module_4_Channel_3_Output"}
	FSOUT_Module_4_Channel_3_Output : BOOL;
	{attribute addProperty Name "FSOUT_Module_4_Channel_4_Output"}
	FSOUT_Module_4_Channel_4_Output : BOOL;
	{attribute addProperty Name "FSOUT_Module_4_ErrAck"}
	FSOUT_Module_4_ErrAck : BOOL;
	{attribute addProperty Name "FSOUT_Module_5_Channel_1_Output"}
	FSOUT_Module_5_Channel_1_Output : BOOL;
	{attribute addProperty Name "FSOUT_Module_5_Channel_2_Output"}
	FSOUT_Module_5_Channel_2_Output : BOOL;
	{attribute addProperty Name "FSOUT_Module_5_Channel_3_Output"}
	FSOUT_Module_5_Channel_3_Output : BOOL;
	{attribute addProperty Name "FSOUT_Module_5_Channel_4_Output"}
	FSOUT_Module_5_Channel_4_Output : BOOL;
	{attribute addProperty Name "FSOUT_Module_5_ErrAck"}
	FSOUT_Module_5_ErrAck : BOOL;
	{attribute addProperty Name "FSOUT_Module_6_Channel_1_Output"}
	FSOUT_Module_6_Channel_1_Output : BOOL;
	{attribute addProperty Name "FSOUT_Module_6_Channel_2_Output"}
	FSOUT_Module_6_Channel_2_Output : BOOL;
	{attribute addProperty Name "FSOUT_Module_6_Channel_3_Output"}
	FSOUT_Module_6_Channel_3_Output : BOOL;
	{attribute addProperty Name "FSOUT_Module_6_Channel_4_Output"}
	FSOUT_Module_6_Channel_4_Output : BOOL;
	{attribute addProperty Name "FSOUT_Module_6_ErrAck"}
	FSOUT_Module_6_ErrAck : BOOL;
	{attribute addProperty Name "FSoE_CRC_001"}
	FSoE_CRC_001 : UINT;
	{attribute addProperty Name "FSIN_Module_1_ErrAck"}
	FSIN_Module_1_ErrAck : BOOL;
	{attribute addProperty Name "FSIN_Module_2_ErrAck"}
	FSIN_Module_2_ErrAck : BOOL;
	{attribute addProperty Name "FSIN_Module_3_ErrAck"}
	FSIN_Module_3_ErrAck : BOOL;
	{attribute addProperty Name "FSIN_Module_4_ErrAck"}
	FSIN_Module_4_ErrAck : BOOL;
	{attribute addProperty Name "FSIN_Module_5_ErrAck"}
	FSIN_Module_5_ErrAck : BOOL;
	{attribute addProperty Name "FSIN_Module_6_ErrAck"}
	FSIN_Module_6_ErrAck : BOOL;
	{attribute addProperty Name "FSIN_Module_7_ErrAck"}
	FSIN_Module_7_ErrAck : BOOL;
	{attribute addProperty Name "FSIN_Module_8_ErrAck"}
	FSIN_Module_8_ErrAck : BOOL;
	{attribute addProperty Name "FSIN_Module_9_ErrAck_1"}
	FSIN_Module_9_ErrAck_1 : BOOL;
	{attribute addProperty Name "FSIN_Module_9_ErrAck_2"}
	FSIN_Module_9_ErrAck_2 : BOOL;
	{attribute addProperty Name "FSIN_Module_10_ErrAck_1"}
	FSIN_Module_10_ErrAck_1 : BOOL;
	{attribute addProperty Name "FSIN_Module_10_ErrAck_2"}
	FSIN_Module_10_ErrAck_2 : BOOL;
	{attribute addProperty Name "FSoE_CRC_002"}
	FSoE_CRC_002 : UINT;
	{attribute addProperty Name "FSoE_Connection_ID"}
	FSoE_Connection_ID : UINT;
END_STRUCT
END_TYPE

// ---- DUTs/IO/PdoEntries/FSOE_39DE0EE0.TcDUT
{attribute 'GeneratedUsingTerminal: EK1960-0000-0021'}
{attribute addProperty BoxType "EK1960-0000-0021"}
{attribute addProperty Id "FSoE_CommandUSINT1FSOUT_Module_1_Module_FaultBOOL1FSOUT_Module_2_Module_FaultBOOL1FSOUT_Module_3_Module_FaultBOOL1FSOUT_Module_4_Module_FaultBOOL1FSOUT_Module_5_Module_FaultBOOL1FSOUT_Module_6_Module_FaultBOOL1FSIN_Module_1_Channel_1_Input_X6_1BOOL1FSIN_Module_1_Channel_2_Input_X6_2BOOL1FSIN_Module_1_Module_FaultBOOL1FSIN_Module_2_Channel_1_Input_X6_3BOOL1FSIN_Module_2_Channel_2_Input_X6_4BOOL1FSIN_Module_2_Module_FaultBOOL1FSIN_Module_3_Channel_1_Input_X6_5BOOL1FSIN_Module_3_Channel_2_Input_X6_6BOOL1FSIN_Module_3_Module_FaultBOOL1FSoE_CRC_000UINT2FSIN_Module_4_Channel_1_Input_X6_7BOOL1FSIN_Module_4_Channel_2_Input_X6_8BOOL1FSIN_Module_4_Module_FaultBOOL1FSIN_Module_5_Channel_1_Input_X6_9BOOL1FSIN_Module_5_Channel_2_Input_X6_10BOOL1FSIN_Module_5_Module_FaultBOOL1FSIN_Module_6_Channel_1_Input_X8_1BOOL1FSIN_Module_6_Channel_2_Input_X8_2BOOL1FSIN_Module_6_Module_FaultBOOL1FSIN_Module_7_Channel_1_Input_X8_3BOOL1FSIN_Module_7_Channel_2_Input_X8_4BOOL1FSIN_Module_7_Module_FaultBOOL1FSIN_Module_8_Channel_1_Input_X8_5BOOL1FSIN_Module_8_Channel_2_Input_X8_6BOOL1FSIN_Module_8_Module_FaultBOOL1FSIN_Module_9_Channel_1_Input_X8_7BOOL1FSoE_CRC_001UINT2FSIN_Module_9_Channel_2_Input_X8_8BOOL1FSIN_Module_9_Module_Fault_1BOOL1FSIN_Module_9_Module_Fault_2BOOL1FSIN_Module_10_Channel_1_Input_X8_9BOOL1FSIN_Module_10_Channel_2_Input_X8_10BOOL1FSIN_Module_10_Module_Fault_1BOOL1FSIN_Module_10_Module_Fault_2BOOL1FSoE_CRC_002UINT2FSoE_Connection_IDUINT2"}
{attribute addProperty CRC "970854112"}
{attribute addProperty Size "47"}
TYPE FSOE_39DE0EE0 :
STRUCT
	{attribute addProperty Name "FSoE_Command"}
	FSoE_Command : USINT;
	{attribute addProperty Name "FSOUT_Module_1_Module_Fault"}
	FSOUT_Module_1_Module_Fault : BOOL;
	{attribute addProperty Name "FSOUT_Module_2_Module_Fault"}
	FSOUT_Module_2_Module_Fault : BOOL;
	{attribute addProperty Name "FSOUT_Module_3_Module_Fault"}
	FSOUT_Module_3_Module_Fault : BOOL;
	{attribute addProperty Name "FSOUT_Module_4_Module_Fault"}
	FSOUT_Module_4_Module_Fault : BOOL;
	{attribute addProperty Name "FSOUT_Module_5_Module_Fault"}
	FSOUT_Module_5_Module_Fault : BOOL;
	{attribute addProperty Name "FSOUT_Module_6_Module_Fault"}
	FSOUT_Module_6_Module_Fault : BOOL;
	{attribute addProperty Name "FSIN_Module_1_Channel_1_Input_X6_1"}
	FSIN_Module_1_Channel_1_Input_X6_1 : BOOL;
	{attribute addProperty Name "FSIN_Module_1_Channel_2_Input_X6_2"}
	FSIN_Module_1_Channel_2_Input_X6_2 : BOOL;
	{attribute addProperty Name "FSIN_Module_1_Module_Fault"}
	FSIN_Module_1_Module_Fault : BOOL;
	{attribute addProperty Name "FSIN_Module_2_Channel_1_Input_X6_3"}
	FSIN_Module_2_Channel_1_Input_X6_3 : BOOL;
	{attribute addProperty Name "FSIN_Module_2_Channel_2_Input_X6_4"}
	FSIN_Module_2_Channel_2_Input_X6_4 : BOOL;
	{attribute addProperty Name "FSIN_Module_2_Module_Fault"}
	FSIN_Module_2_Module_Fault : BOOL;
	{attribute addProperty Name "FSIN_Module_3_Channel_1_Input_X6_5"}
	FSIN_Module_3_Channel_1_Input_X6_5 : BOOL;
	{attribute addProperty Name "FSIN_Module_3_Channel_2_Input_X6_6"}
	FSIN_Module_3_Channel_2_Input_X6_6 : BOOL;
	{attribute addProperty Name "FSIN_Module_3_Module_Fault"}
	FSIN_Module_3_Module_Fault : BOOL;
	{attribute addProperty Name "FSoE_CRC_000"}
	FSoE_CRC_000 : UINT;
	{attribute addProperty Name "FSIN_Module_4_Channel_1_Input_X6_7"}
	FSIN_Module_4_Channel_1_Input_X6_7 : BOOL;
	{attribute addProperty Name "FSIN_Module_4_Channel_2_Input_X6_8"}
	FSIN_Module_4_Channel_2_Input_X6_8 : BOOL;
	{attribute addProperty Name "FSIN_Module_4_Module_Fault"}
	FSIN_Module_4_Module_Fault : BOOL;
	{attribute addProperty Name "FSIN_Module_5_Channel_1_Input_X6_9"}
	FSIN_Module_5_Channel_1_Input_X6_9 : BOOL;
	{attribute addProperty Name "FSIN_Module_5_Channel_2_Input_X6_10"}
	FSIN_Module_5_Channel_2_Input_X6_10 : BOOL;
	{attribute addProperty Name "FSIN_Module_5_Module_Fault"}
	FSIN_Module_5_Module_Fault : BOOL;
	{attribute addProperty Name "FSIN_Module_6_Channel_1_Input_X8_1"}
	FSIN_Module_6_Channel_1_Input_X8_1 : BOOL;
	{attribute addProperty Name "FSIN_Module_6_Channel_2_Input_X8_2"}
	FSIN_Module_6_Channel_2_Input_X8_2 : BOOL;
	{attribute addProperty Name "FSIN_Module_6_Module_Fault"}
	FSIN_Module_6_Module_Fault : BOOL;
	{attribute addProperty Name "FSIN_Module_7_Channel_1_Input_X8_3"}
	FSIN_Module_7_Channel_1_Input_X8_3 : BOOL;
	{attribute addProperty Name "FSIN_Module_7_Channel_2_Input_X8_4"}
	FSIN_Module_7_Channel_2_Input_X8_4 : BOOL;
	{attribute addProperty Name "FSIN_Module_7_Module_Fault"}
	FSIN_Module_7_Module_Fault : BOOL;
	{attribute addProperty Name "FSIN_Module_8_Channel_1_Input_X8_5"}
	FSIN_Module_8_Channel_1_Input_X8_5 : BOOL;
	{attribute addProperty Name "FSIN_Module_8_Channel_2_Input_X8_6"}
	FSIN_Module_8_Channel_2_Input_X8_6 : BOOL;
	{attribute addProperty Name "FSIN_Module_8_Module_Fault"}
	FSIN_Module_8_Module_Fault : BOOL;
	{attribute addProperty Name "FSIN_Module_9_Channel_1_Input_X8_7"}
	FSIN_Module_9_Channel_1_Input_X8_7 : BOOL;
	{attribute addProperty Name "FSoE_CRC_001"}
	FSoE_CRC_001 : UINT;
	{attribute addProperty Name "FSIN_Module_9_Channel_2_Input_X8_8"}
	FSIN_Module_9_Channel_2_Input_X8_8 : BOOL;
	{attribute addProperty Name "FSIN_Module_9_Module_Fault_1"}
	FSIN_Module_9_Module_Fault_1 : BOOL;
	{attribute addProperty Name "FSIN_Module_9_Module_Fault_2"}
	FSIN_Module_9_Module_Fault_2 : BOOL;
	{attribute addProperty Name "FSIN_Module_10_Channel_1_Input_X8_9"}
	FSIN_Module_10_Channel_1_Input_X8_9 : BOOL;
	{attribute addProperty Name "FSIN_Module_10_Channel_2_Input_X8_10"}
	FSIN_Module_10_Channel_2_Input_X8_10 : BOOL;
	{attribute addProperty Name "FSIN_Module_10_Module_Fault_1"}
	FSIN_Module_10_Module_Fault_1 : BOOL;
	{attribute addProperty Name "FSIN_Module_10_Module_Fault_2"}
	FSIN_Module_10_Module_Fault_2 : BOOL;
	{attribute addProperty Name "FSoE_CRC_002"}
	FSoE_CRC_002 : UINT;
	{attribute addProperty Name "FSoE_Connection_ID"}
	FSoE_Connection_ID : UINT;
END_STRUCT
END_TYPE

// ---- DUTs/IO/PdoEntries/FSOE_3E4279E1.TcDUT
{attribute 'GeneratedUsingTerminal: EK1960-0000-0021'}
{attribute addProperty BoxType "EK1960-0000-0021"}
{attribute addProperty Id "FSoE_CommandUSINT1FSOUT_Module_1_Channel_1_Output_X5_1BOOL1FSOUT_Module_1_Channel_2_Output_X5_2BOOL1FSOUT_Module_1_Channel_3_Output_X5_3BOOL1FSOUT_Module_1_Channel_4_Output_X5_4BOOL1FSOUT_Module_1_ErrAckBOOL1FSOUT_Module_2_Channel_1_Output_X5_5BOOL1FSOUT_Module_2_Channel_2_Output_X5_6BOOL1FSOUT_Module_2_Channel_3_Output_X5_7BOOL1FSOUT_Module_2_Channel_4_Output_X5_8BOOL1FSOUT_Module_2_ErrAckBOOL1FSOUT_Module_3_Channel_1_Output_X7_1BOOL1FSOUT_Module_3_Channel_2_Output_X7_2BOOL1FSOUT_Module_3_Channel_3_Output_X7_3BOOL1FSOUT_Module_3_Channel_4_Output_X7_4BOOL1FSOUT_Module_3_ErrAckBOOL1FSOUT_Module_4_Channel_1_Output_X7_5BOOL1FSoE_CRC_000UINT2FSOUT_Module_4_Channel_2_Output_X7_6BOOL1FSOUT_Module_4_Channel_3_Output_X7_7BOOL1FSOUT_Module_4_Channel_4_Output_X7_8BOOL1FSOUT_Module_4_ErrAckBOOL1FSOUT_Module_5_Channel_1_Output_X9_1BOOL1FSOUT_Module_5_Channel_2_Output_X9_2BOOL1FSOUT_Module_5_Channel_3_Output_X9_3BOOL1FSOUT_Module_5_Channel_4_Output_X9_4BOOL1FSOUT_Module_5_ErrAckBOOL1FSOUT_Module_6_Channel_1_Output_X9_5BOOL1FSOUT_Module_6_Channel_2_Output_X9_6BOOL1FSOUT_Module_6_Channel_3_Output_X9_7BOOL1FSOUT_Module_6_Channel_4_Output_X9_8BOOL1FSOUT_Module_6_ErrAckBOOL1FSoE_CRC_001UINT2FSIN_Module_1_ErrAckBOOL1FSIN_Module_2_ErrAckBOOL1FSIN_Module_3_ErrAckBOOL1FSIN_Module_4_ErrAckBOOL1FSIN_Module_5_ErrAckBOOL1FSIN_Module_6_ErrAckBOOL1FSIN_Module_7_ErrAckBOOL1FSIN_Module_8_ErrAckBOOL1FSIN_Module_9_Err_Ack_1BOOL1FSIN_Module_9_Err_Ack_2BOOL1FSIN_Module_10_Err_Ack_1BOOL1FSIN_Module_10_Err_Ack_2BOOL1FSoE_CRC_002UINT2FSoE_Connection_IDUINT2"}
{attribute addProperty CRC "1044543969"}
{attribute addProperty Size "51"}
TYPE FSOE_3E4279E1 :
STRUCT
	{attribute addProperty Name "FSoE_Command"}
	FSoE_Command : USINT;
	{attribute addProperty Name "FSOUT_Module_1_Channel_1_Output_X5_1"}
	FSOUT_Module_1_Channel_1_Output_X5_1 : BOOL;
	{attribute addProperty Name "FSOUT_Module_1_Channel_2_Output_X5_2"}
	FSOUT_Module_1_Channel_2_Output_X5_2 : BOOL;
	{attribute addProperty Name "FSOUT_Module_1_Channel_3_Output_X5_3"}
	FSOUT_Module_1_Channel_3_Output_X5_3 : BOOL;
	{attribute addProperty Name "FSOUT_Module_1_Channel_4_Output_X5_4"}
	FSOUT_Module_1_Channel_4_Output_X5_4 : BOOL;
	{attribute addProperty Name "FSOUT_Module_1_ErrAck"}
	FSOUT_Module_1_ErrAck : BOOL;
	{attribute addProperty Name "FSOUT_Module_2_Channel_1_Output_X5_5"}
	FSOUT_Module_2_Channel_1_Output_X5_5 : BOOL;
	{attribute addProperty Name "FSOUT_Module_2_Channel_2_Output_X5_6"}
	FSOUT_Module_2_Channel_2_Output_X5_6 : BOOL;
	{attribute addProperty Name "FSOUT_Module_2_Channel_3_Output_X5_7"}
	FSOUT_Module_2_Channel_3_Output_X5_7 : BOOL;
	{attribute addProperty Name "FSOUT_Module_2_Channel_4_Output_X5_8"}
	FSOUT_Module_2_Channel_4_Output_X5_8 : BOOL;
	{attribute addProperty Name "FSOUT_Module_2_ErrAck"}
	FSOUT_Module_2_ErrAck : BOOL;
	{attribute addProperty Name "FSOUT_Module_3_Channel_1_Output_X7_1"}
	FSOUT_Module_3_Channel_1_Output_X7_1 : BOOL;
	{attribute addProperty Name "FSOUT_Module_3_Channel_2_Output_X7_2"}
	FSOUT_Module_3_Channel_2_Output_X7_2 : BOOL;
	{attribute addProperty Name "FSOUT_Module_3_Channel_3_Output_X7_3"}
	FSOUT_Module_3_Channel_3_Output_X7_3 : BOOL;
	{attribute addProperty Name "FSOUT_Module_3_Channel_4_Output_X7_4"}
	FSOUT_Module_3_Channel_4_Output_X7_4 : BOOL;
	{attribute addProperty Name "FSOUT_Module_3_ErrAck"}
	FSOUT_Module_3_ErrAck : BOOL;
	{attribute addProperty Name "FSOUT_Module_4_Channel_1_Output_X7_5"}
	FSOUT_Module_4_Channel_1_Output_X7_5 : BOOL;
	{attribute addProperty Name "FSoE_CRC_000"}
	FSoE_CRC_000 : UINT;
	{attribute addProperty Name "FSOUT_Module_4_Channel_2_Output_X7_6"}
	FSOUT_Module_4_Channel_2_Output_X7_6 : BOOL;
	{attribute addProperty Name "FSOUT_Module_4_Channel_3_Output_X7_7"}
	FSOUT_Module_4_Channel_3_Output_X7_7 : BOOL;
	{attribute addProperty Name "FSOUT_Module_4_Channel_4_Output_X7_8"}
	FSOUT_Module_4_Channel_4_Output_X7_8 : BOOL;
	{attribute addProperty Name "FSOUT_Module_4_ErrAck"}
	FSOUT_Module_4_ErrAck : BOOL;
	{attribute addProperty Name "FSOUT_Module_5_Channel_1_Output_X9_1"}
	FSOUT_Module_5_Channel_1_Output_X9_1 : BOOL;
	{attribute addProperty Name "FSOUT_Module_5_Channel_2_Output_X9_2"}
	FSOUT_Module_5_Channel_2_Output_X9_2 : BOOL;
	{attribute addProperty Name "FSOUT_Module_5_Channel_3_Output_X9_3"}
	FSOUT_Module_5_Channel_3_Output_X9_3 : BOOL;
	{attribute addProperty Name "FSOUT_Module_5_Channel_4_Output_X9_4"}
	FSOUT_Module_5_Channel_4_Output_X9_4 : BOOL;
	{attribute addProperty Name "FSOUT_Module_5_ErrAck"}
	FSOUT_Module_5_ErrAck : BOOL;
	{attribute addProperty Name "FSOUT_Module_6_Channel_1_Output_X9_5"}
	FSOUT_Module_6_Channel_1_Output_X9_5 : BOOL;
	{attribute addProperty Name "FSOUT_Module_6_Channel_2_Output_X9_6"}
	FSOUT_Module_6_Channel_2_Output_X9_6 : BOOL;
	{attribute addProperty Name "FSOUT_Module_6_Channel_3_Output_X9_7"}
	FSOUT_Module_6_Channel_3_Output_X9_7 : BOOL;
	{attribute addProperty Name "FSOUT_Module_6_Channel_4_Output_X9_8"}
	FSOUT_Module_6_Channel_4_Output_X9_8 : BOOL;
	{attribute addProperty Name "FSOUT_Module_6_ErrAck"}
	FSOUT_Module_6_ErrAck : BOOL;
	{attribute addProperty Name "FSoE_CRC_001"}
	FSoE_CRC_001 : UINT;
	{attribute addProperty Name "FSIN_Module_1_ErrAck"}
	FSIN_Module_1_ErrAck : BOOL;
	{attribute addProperty Name "FSIN_Module_2_ErrAck"}
	FSIN_Module_2_ErrAck : BOOL;
	{attribute addProperty Name "FSIN_Module_3_ErrAck"}
	FSIN_Module_3_ErrAck : BOOL;
	{attribute addProperty Name "FSIN_Module_4_ErrAck"}
	FSIN_Module_4_ErrAck : BOOL;
	{attribute addProperty Name "FSIN_Module_5_ErrAck"}
	FSIN_Module_5_ErrAck : BOOL;
	{attribute addProperty Name "FSIN_Module_6_ErrAck"}
	FSIN_Module_6_ErrAck : BOOL;
	{attribute addProperty Name "FSIN_Module_7_ErrAck"}
	FSIN_Module_7_ErrAck : BOOL;
	{attribute addProperty Name "FSIN_Module_8_ErrAck"}
	FSIN_Module_8_ErrAck : BOOL;
	{attribute addProperty Name "FSIN_Module_9_Err_Ack_1"}
	FSIN_Module_9_Err_Ack_1 : BOOL;
	{attribute addProperty Name "FSIN_Module_9_Err_Ack_2"}
	FSIN_Module_9_Err_Ack_2 : BOOL;
	{attribute addProperty Name "FSIN_Module_10_Err_Ack_1"}
	FSIN_Module_10_Err_Ack_1 : BOOL;
	{attribute addProperty Name "FSIN_Module_10_Err_Ack_2"}
	FSIN_Module_10_Err_Ack_2 : BOOL;
	{attribute addProperty Name "FSoE_CRC_002"}
	FSoE_CRC_002 : UINT;
	{attribute addProperty Name "FSoE_Connection_ID"}
	FSoE_Connection_ID : UINT;
END_STRUCT
END_TYPE

